  MoveL 9308 to (-40.61, 150.52, 135.08) mm, rotated rx 180 ry 0 rz -180 deg; joints [-126.331, -50.727, -84.518, 62.425, 65.347, -38.616]
  Call Extruder(4.93416)
  MoveL 9309 to (-40.66, 150.21, 135.08) mm, rotated rx 180 ry 0 rz -180 deg; joints [-126.35, -50.704, -84.571, 62.397, 65.348, -38.58]
  MoveL 9310 to (-40.66, 150.21, 135.08) mm, rotated rx 180 ry 0 rz -180 deg; joints [-126.35, -50.704, -84.571, 62.397, 65.348, -38.58]
  Call Extruder(5.09479)
  MoveL 9311 to (-40.71, 149.91, 135.08) mm, rotated rx -180 ry 0 rz 180 deg; joints [-126.369, -50.681, -84.624, 62.368, 65.35, -38.544]
  MoveL 9312 to (-40.71, 149.91, 135.08) mm, rotated rx -180 ry 0 rz 180 deg; joints [-126.369, -50.681, -84.624, 62.368, 65.35, -38.544]
  Call Extruder(5.25470)
  MoveL 9313 to (-40.76, 149.6, 135.08) mm, rotated rx 180 ry 0 rz -180 deg; joints [-126.388, -50.658, -84.676, 62.34, 65.352, -38.509]
  MoveL 9314 to (-40.76, 149.6, 135.08) mm, rotated rx 180 ry 0 rz -180 deg; joints [-126.388, -50.658, -84.676, 62.34, 65.352, -38.509]
  Call Extruder(5.41388)
  MoveL 9315 to (-40.81, 149.3, 135.08) mm, rotated rx 180 ry 0 rz 180 deg; joints [-126.407, -50.634, -84.729, 62.311, 65.354, -38.473]
  MoveL 9316 to (-40.81, 149.3, 135.08) mm, rotated rx 180 ry 0 rz 180 deg; joints [-126.407, -50.634, -84.729, 62.311, 65.354, -38.473]
  Call Extruder(5.57233)
  MoveL 9317 to (-40.86, 148.99, 135.08) mm, rotated rx 180 ry 0 rz -180 deg; joints [-126.426, -50.611, -84.782, 62.283, 65.356, -38.437]
  MoveL 9318 to (-40.86, 148.99, 135.08) mm, rotated rx 180 ry 0 rz -180 deg; joints [-126.426, -50.611, -84.782, 62.283, 65.356, -38.437]
  Call Extruder(5.77120)
  MoveL 9319 to (-40.9, 148.6, 135.08) mm, rotated rx 180 ry 0 rz 180 deg; joints [-126.452, -50.583, -84.847, 62.246, 65.357, -38.393]
  MoveL 9320 to (-40.9, 148.6, 135.08) mm, rotated rx 180 ry 0 rz 180 deg; joints [-126.452, -50.583, -84.847, 62.246, 65.357, -38.393]
  Call Extruder(5.96921)
  MoveL 9321 to (-40.95, 148.22, 135.08) mm, rotated rx 180 ry 0 rz 180 deg; joints [-126.478, -50.554, -84.912, 62.208, 65.358, -38.348]
  MoveL 9322 to (-40.95, 148.22, 135.08) mm, rotated rx 180 ry 0 rz 180 deg; joints [-126.478, -50.554, -84.912, 62.208, 65.358, -38.348]
  Call Extruder(6.16635)
  MoveL 9323 to (-40.99, 147.83, 135.08) mm, rotated rx 180 ry 0 rz -180 deg; joints [-126.504, -50.526, -84.977, 62.171, 65.359, -38.303]
  MoveL 9324 to (-40.99, 147.83, 135.08) mm, rotated rx 180 ry 0 rz -180 deg; joints [-126.504, -50.526, -84.977, 62.171, 65.359, -38.303]
  Call Extruder(6.36262)
  MoveL 9325 to (-41.04, 147.44, 135.08) mm, rotated rx -180 ry 0 rz 180 deg; joints [-126.53, -50.498, -85.041, 62.134, 65.359, -38.258]
  MoveL 9326 to (-41.04, 147.44, 135.08) mm, rotated rx -180 ry 0 rz 180 deg; joints [-126.53, -50.498, -85.041, 62.134, 65.359, -38.258]
  Call Extruder(6.60831)
  MoveL 9327 to (-41.09, 146.95, 135.08) mm, rotated rx 180 ry 0 rz 180 deg; joints [-126.564, -50.462, -85.122, 62.086, 65.359, -38.202]
  MoveL 9328 to (-41.09, 146.95, 135.08) mm, rotated rx 180 ry 0 rz 180 deg; joints [-126.564, -50.462, -85.122, 62.086, 65.359, -38.202]
  Call Extruder(6.90304)
  MoveL 9329 to (-41.13, 146.36, 135.08) mm, rotated rx 180 ry 0 rz 180 deg; joints [-126.607, -50.421, -85.217, 62.028, 65.358, -38.134]
  MoveL 9330 to (-41.13, 146.36, 135.08) mm, rotated rx 180 ry 0 rz 180 deg; joints [-126.607, -50.421, -85.217, 62.028, 65.358, -38.134]
  Call Extruder(7.19644)
  MoveL 9331 to (-41.18, 145.77, 135.08) mm, rotated rx 180 ry 0 rz -180 deg; joints [-126.649, -50.379, -85.313, 61.969, 65.358, -38.067]
  MoveL 9332 to (-41.18, 145.77, 135.08) mm, rotated rx 180 ry 0 rz -180 deg; joints [-126.649, -50.379, -85.313, 61.969, 65.358, -38.067]
  Call Extruder(7.62977)
  MoveL 9333 to (-41.22, 144.9, 135.08) mm, rotated rx -180 ry 0 rz -180 deg; joints [-126.715, -50.318, -85.452, 61.881, 65.354, -37.967]
  MoveL 9334 to (-41.22, 144.9, 135.08) mm, rotated rx -180 ry 0 rz -180 deg; joints [-126.715, -50.318, -85.452, 61.881, 65.354, -37.967]
  Call Extruder(8.20193)
  MoveL 9335 to (-41.27, 143.74, 135.08) mm, rotated rx 180 ry 0 rz 180 deg; joints [-126.804, -50.238, -85.635, 61.762, 65.348, -37.835]
  MoveL 9336 to (-41.27, 143.74, 135.08) mm, rotated rx 180 ry 0 rz 180 deg; joints [-126.804, -50.238, -85.635, 61.762, 65.348, -37.835]
  Call Extruder(8.62976)
  MoveL 9337 to (-41.29, 142.86, 135.08) mm, rotated rx -180 ry 0 rz 180 deg; joints [-126.873, -50.179, -85.77, 61.671, 65.341, -37.736]
  Call Extruder(50.62329)
  MoveL 9338 to (-41.29, 57.14, 135.08) mm, rotated rx 180 ry 0 rz 180 deg; joints [-135.148, -45.231, -97.556, 51.322, 64.612, -28.173]
  MoveL 9339 to (-41.29, 57.14, 135.08) mm, rotated rx 180 ry 0 rz 180 deg; joints [-135.148, -45.231, -97.556, 51.322, 64.612, -28.173]
  Call Extruder(51.33886)
  MoveL 9340 to (-41.25, 55.68, 135.08) mm, rotated rx -180 ry 0 rz 180 deg; joints [-135.318, -45.162, -97.729, 51.117, 64.597, -28.012]
  MoveL 9341 to (-41.25, 55.68, 135.08) mm, rotated rx -180 ry 0 rz 180 deg; joints [-135.318, -45.162, -97.729, 51.117, 64.597, -28.012]
  Call Extruder(51.91360)
  MoveL 9342 to (-41.2, 54.52, 135.08) mm, rotated rx 180 ry 0 rz -180 deg; joints [-135.457, -45.107, -97.865, 50.952, 64.583, -27.884]
  MoveL 9343 to (-41.2, 54.52, 135.08) mm, rotated rx 180 ry 0 rz -180 deg; joints [-135.457, -45.107, -97.865, 50.952, 64.583, -27.884]
  Call Extruder(52.20698)
  MoveL 9344 to (-41.15, 53.93, 135.08) mm, rotated rx 180 ry 0 rz 180 deg; joints [-135.53, -45.081, -97.932, 50.866, 64.574, -27.819]
  MoveL 9345 to (-41.15, 53.93, 135.08) mm, rotated rx 180 ry 0 rz 180 deg; joints [-135.53, -45.081, -97.932, 50.866, 64.574, -27.819]
  Call Extruder(52.50168)
  MoveL 9346 to (-41.11, 53.34, 135.08) mm, rotated rx 180 ry 0 rz -180 deg; joints [-135.603, -45.054, -97.997, 50.779, 64.565, -27.754]
  MoveL 9347 to (-41.11, 53.34, 135.08) mm, rotated rx 180 ry 0 rz -180 deg; joints [-135.603, -45.054, -97.997, 50.779, 64.565, -27.754]
  Call Extruder(52.79772)
  MoveL 9348 to (-41.06, 52.75, 135.08) mm, rotated rx -180 ry 0 rz 180 deg; joints [-135.676, -45.028, -98.063, 50.693, 64.556, -27.689]
  MoveL 9349 to (-41.06, 52.75, 135.08) mm, rotated rx -180 ry 0 rz 180 deg; joints [-135.676, -45.028, -98.063, 50.693, 64.556, -27.689]
  Call Extruder(52.99180)
  MoveL 9350 to (-41.02, 52.37, 135.08) mm, rotated rx -180 ry 0 rz 180 deg; joints [-135.726, -45.012, -98.104, 50.635, 64.549, -27.647]
  MoveL 9351 to (-41.02, 52.37, 135.08) mm, rotated rx -180 ry 0 rz 180 deg; joints [-135.726, -45.012, -98.104, 50.635, 64.549, -27.647]
  Call Extruder(53.18958)
  MoveL 9352 to (-40.97, 51.98, 135.08) mm, rotated rx 180 ry 0 rz -180 deg; joints [-135.776, -44.995, -98.145, 50.577, 64.541, -27.605]
  MoveL 9353 to (-40.97, 51.98, 135.08) mm, rotated rx 180 ry 0 rz -180 deg; joints [-135.776, -44.995, -98.145, 50.577, 64.541, -27.605]
  Call Extruder(53.38824)
  MoveL 9354 to (-40.92, 51.59, 135.08) mm, rotated rx 180 ry 0 rz 180 deg; joints [-135.826, -44.979, -98.187, 50.518, 64.534, -27.562]
  MoveL 9355 to (-40.92, 51.59, 135.08) mm, rotated rx 180 ry 0 rz 180 deg; joints [-135.826, -44.979, -98.187, 50.518, 64.534, -27.562]
  Call Extruder(53.58777)
  MoveL 9356 to (-40.88, 51.2, 135.08) mm, rotated rx 180 ry 0 rz -180 deg; joints [-135.877, -44.963, -98.228, 50.46, 64.526, -27.52]
  MoveL 9357 to (-40.88, 51.2, 135.08) mm, rotated rx 180 ry 0 rz -180 deg; joints [-135.877, -44.963, -98.228, 50.46, 64.526, -27.52]
  Call Extruder(53.76717)
  MoveL 9358 to (-40.83, 50.86, 135.08) mm, rotated rx 180 ry 0 rz -180 deg; joints [-135.922, -44.948, -98.264, 50.407, 64.519, -27.482]
  MoveL 9359 to (-40.83, 50.86, 135.08) mm, rotated rx 180 ry 0 rz -180 deg; joints [-135.922, -44.948, -98.264, 50.407, 64.519, -27.482]
  Call Extruder(53.92635)
  MoveL 9360 to (-40.78, 50.55, 135.08) mm, rotated rx -180 ry 0 rz -180 deg; joints [-135.964, -44.936, -98.295, 50.36, 64.512, -27.449]
  MoveL 9361 to (-40.78, 50.55, 135.08) mm, rotated rx -180 ry 0 rz -180 deg; joints [-135.964, -44.936, -98.295, 50.36, 64.512, -27.449]
  Call Extruder(54.08625)
  MoveL 9362 to (-40.73, 50.24, 135.08) mm, rotated rx -180 ry 0 rz -180 deg; joints [-136.005, -44.924, -98.326, 50.312, 64.504, -27.416]
  MoveL 9363 to (-40.73, 50.24, 135.08) mm, rotated rx -180 ry 0 rz -180 deg; joints [-136.005, -44.924, -98.326, 50.312, 64.504, -27.416]
  Call Extruder(54.24689)
  MoveL 9364 to (-40.69, 49.94, 135.08) mm, rotated rx 180 ry 0 rz -180 deg; joints [-136.046, -44.911, -98.356, 50.265, 64.497, -27.382]
  MoveL 9365 to (-40.69, 49.94, 135.08) mm, rotated rx 180 ry 0 rz -180 deg; joints [-136.046, -44.911, -98.356, 50.265, 64.497, -27.382]
  Call Extruder(54.40825)
  MoveL 9366 to (-40.64, 49.63, 135.08) mm, rotated rx 180 ry 0 rz 180 deg; joints [-136.087, -44.899, -98.387, 50.218, 64.49, -27.349]
  MoveL 9367 to (-40.64, 49.63, 135.08) mm, rotated rx 180 ry 0 rz 180 deg; joints [-136.087, -44.899, -98.387, 50.218, 64.49, -27.349]
  Call Extruder(54.57034)
  MoveL 9368 to (-40.59, 49.33, 135.08) mm, rotated rx 180 ry 0 rz -180 deg; joints [-136.128, -44.887, -98.418, 50.17, 64.483, -27.316]
  MoveL 9369 to (-40.59, 49.33, 135.08) mm, rotated rx 180 ry 0 rz -180 deg; joints [-136.128, -44.887, -98.418, 50.17, 64.483, -27.316]
  Call Extruder(54.71853)
  MoveL 9370 to (-40.54, 49.05, 135.08) mm, rotated rx -180 ry 0 rz 180 deg; joints [-136.166, -44.876, -98.445, 50.127, 64.476, -27.286]
  MoveL 9371 to (-40.54, 49.05, 135.08) mm, rotated rx -180 ry 0 rz 180 deg; joints [-136.166, -44.876, -98.445, 50.127, 64.476, -27.286]
  Call Extruder(54.85276)
  MoveL 9372 to (-40.49, 48.8, 135.08) mm, rotated rx 180 ry 0 rz -180 deg; joints [-136.201, -44.867, -98.468, 50.087, 64.469, -27.259]
  MoveL 9373 to (-40.49, 48.8, 135.08) mm, rotated rx 180 ry 0 rz -180 deg; joints [-136.201, -44.867, -98.468, 50.087, 64.469, -27.259]
  Call Extruder(54.98760)
  MoveL 9374 to (-40.44, 48.55, 135.08) mm, rotated rx 180 ry 0 rz -180 deg; joints [-136.236, -44.858, -98.492, 50.048, 64.462, -27.232]
  MoveL 9375 to (-40.44, 48.55, 135.08) mm, rotated rx 180 ry 0 rz -180 deg; joints [-136.236, -44.858, -98.492, 50.048, 64.462, -27.232]
  Call Extruder(55.12305)
  MoveL 9376 to (-40.39, 48.3, 135.08) mm, rotated rx 180 ry 0 rz 180 deg; joints [-136.271, -44.848, -98.516, 50.008, 64.456, -27.205]
  MoveL 9377 to (-40.39, 48.3, 135.08) mm, rotated rx 180 ry 0 rz 180 deg; joints [-136.271, -44.848, -98.516, 50.008, 64.456, -27.205]
  Call Extruder(55.25911)
  MoveL 9378 to (-40.34, 48.05, 135.08) mm, rotated rx -180 ry 0 rz 180 deg; joints [-136.306, -44.839, -98.539, 49.969, 64.449, -27.178]
  MoveL 9379 to (-40.34, 48.05, 135.08) mm, rotated rx -180 ry 0 rz 180 deg; joints [-136.306, -44.839, -98.539, 49.969, 64.449, -27.178]
  Call Extruder(55.39578)
  MoveL 9380 to (-40.29, 47.8, 135.08) mm, rotated rx -180 ry 0 rz -180 deg; joints [-136.341, -44.829, -98.563, 49.929, 64.442, -27.151]
  MoveL 9381 to (-40.29, 47.8, 135.08) mm, rotated rx -180 ry 0 rz -180 deg; joints [-136.341, -44.829, -98.563, 49.929, 64.442, -27.151]
  Call Extruder(55.53306)
  MoveL 9382 to (-40.24, 47.55, 135.08) mm, rotated rx -180 ry 0 rz -180 deg; joints [-136.376, -44.82, -98.586, 49.889, 64.435, -27.124]
  MoveL 9383 to (-40.24, 47.55, 135.08) mm, rotated rx -180 ry 0 rz -180 deg; joints [-136.376, -44.82, -98.586, 49.889, 64.435, -27.124]
  Call Extruder(55.65874)
  MoveL 9384 to (-40.2, 47.33, 135.08) mm, rotated rx 180 ry 0 rz 180 deg; joints [-136.408, -44.812, -98.607, 49.853, 64.429, -27.1]
  MoveL 9385 to (-40.2, 47.33, 135.08) mm, rotated rx 180 ry 0 rz 180 deg; joints [-136.408, -44.812, -98.607, 49.853, 64.429, -27.1]
  Call Extruder(55.77269)
  MoveL 9386 to (-40.15, 47.12, 135.08) mm, rotated rx 180 ry 0 rz -180 deg; joints [-136.437, -44.804, -98.626, 49.82, 64.423, -27.078]
  MoveL 9387 to (-40.15, 47.12, 135.08) mm, rotated rx 180 ry 0 rz -180 deg; joints [-136.437, -44.804, -98.626, 49.82, 64.423, -27.078]
  Call Extruder(55.88710)
  MoveL 9388 to (-40.11, 46.92, 135.08) mm, rotated rx 180 ry 0 rz 180 deg; joints [-136.466, -44.797, -98.645, 49.787, 64.417, -27.056]
  MoveL 9389 to (-40.11, 46.92, 135.08) mm, rotated rx 180 ry 0 rz 180 deg; joints [-136.466, -44.797, -98.645, 49.787, 64.417, -27.056]
  Call Extruder(56.00196)
  MoveL 9390 to (-40.06, 46.72, 135.08) mm, rotated rx 180 ry 0 rz 180 deg; joints [-136.495, -44.789, -98.664, 49.754, 64.411, -27.034]
  MoveL 9391 to (-40.06, 46.72, 135.08) mm, rotated rx 180 ry 0 rz 180 deg; joints [-136.495, -44.789, -98.664, 49.754, 64.411, -27.034]
  Call Extruder(56.11727)
  MoveL 9392 to (-40.02, 46.51, 135.08) mm, rotated rx -180 ry 0 rz -180 deg; joints [-136.525, -44.782, -98.682, 49.721, 64.405, -27.012]
  MoveL 9393 to (-40.02, 46.51, 135.08) mm, rotated rx -180 ry 0 rz -180 deg; joints [-136.525, -44.782, -98.682, 49.721, 64.405, -27.012]
  Call Extruder(56.24665)
  MoveL 9394 to (-39.95, 46.29, 135.08) mm, rotated rx 180 ry 0 rz -180 deg; joints [-136.559, -44.775, -98.701, 49.684, 64.397, -26.988]
  MoveL 9395 to (-39.95, 46.29, 135.08) mm, rotated rx 180 ry 0 rz -180 deg; joints [-136.559, -44.775, -98.701, 49.684, 64.397, -26.988]
  Call Extruder(56.37660)
  MoveL 9396 to (-39.88, 46.06, 135.08) mm, rotated rx 180 ry 0 rz -180 deg; joints [-136.593, -44.768, -98.719, 49.646, 64.388, -26.964]
  MoveL 9397 to (-39.88, 46.06, 135.08) mm, rotated rx 180 ry 0 rz -180 deg; joints [-136.593, -44.768, -98.719, 49.646, 64.388, -26.964]
  Call Extruder(56.50711)
  MoveL 9398 to (-39.81, 45.84, 135.08) mm, rotated rx 180 ry 0 rz 180 deg; joints [-136.627, -44.76, -98.737, 49.608, 64.38, -26.941]
  MoveL 9399 to (-39.81, 45.84, 135.08) mm, rotated rx 180 ry 0 rz 180 deg; joints [-136.627, -44.76, -98.737, 49.608, 64.38, -26.941]
  Call Extruder(56.63818)
  MoveL 9400 to (-39.75, 45.62, 135.08) mm, rotated rx -180 ry 0 rz 180 deg; joints [-136.661, -44.753, -98.755, 49.57, 64.371, -26.917]
  MoveL 9401 to (-39.75, 45.62, 135.08) mm, rotated rx -180 ry 0 rz 180 deg; joints [-136.661, -44.753, -98.755, 49.57, 64.371, -26.917]
  Call Extruder(56.75983)
  MoveL 9402 to (-39.68, 45.41, 135.08) mm, rotated rx 180 ry 0 rz -180 deg; joints [-136.693, -44.747, -98.771, 49.535, 64.363, -26.895]
  MoveL 9403 to (-39.68, 45.41, 135.08) mm, rotated rx 180 ry 0 rz -180 deg; joints [-136.693, -44.747, -98.771, 49.535, 64.363, -26.895]
  Call Extruder(56.87195)
  MoveL 9404 to (-39.62, 45.22, 135.08) mm, rotated rx 180 ry 0 rz 180 deg; joints [-136.722, -44.741, -98.786, 49.503, 64.356, -26.875]
  MoveL 9405 to (-39.62, 45.22, 135.08) mm, rotated rx 180 ry 0 rz 180 deg; joints [-136.722, -44.741, -98.786, 49.503, 64.356, -26.875]
  Call Extruder(56.98452)
  MoveL 9406 to (-39.56, 45.03, 135.08) mm, rotated rx 180 ry 0 rz -180 deg; joints [-136.751, -44.735, -98.8, 49.471, 64.348, -26.855]
  MoveL 9407 to (-39.56, 45.03, 135.08) mm, rotated rx 180 ry 0 rz -180 deg; joints [-136.751, -44.735, -98.8, 49.471, 64.348, -26.855]
  Call Extruder(57.09753)
  MoveL 9408 to (-39.5, 44.85, 135.08) mm, rotated rx 180 ry 0 rz -180 deg; joints [-136.781, -44.73, -98.815, 49.439, 64.341, -26.835]
  MoveL 9409 to (-39.5, 44.85, 135.08) mm, rotated rx 180 ry 0 rz -180 deg; joints [-136.781, -44.73, -98.815, 49.439, 64.341, -26.835]
  Call Extruder(57.21099)
  MoveL 9410 to (-39.44, 44.66, 135.08) mm, rotated rx 180 ry 0 rz -180 deg; joints [-136.81, -44.724, -98.829, 49.406, 64.333, -26.815]
  MoveL 9411 to (-39.44, 44.66, 135.08) mm, rotated rx 180 ry 0 rz -180 deg; joints [-136.81, -44.724, -98.829, 49.406, 64.333, -26.815]
  Call Extruder(57.35863)
  MoveL 9412 to (-39.35, 44.42, 135.08) mm, rotated rx 180 ry 0 rz -180 deg; joints [-136.849, -44.717, -98.846, 49.364, 64.322, -26.79]
  MoveL 9413 to (-39.35, 44.42, 135.08) mm, rotated rx 180 ry 0 rz -180 deg; joints [-136.849, -44.717, -98.846, 49.364, 64.322, -26.79]
  Call Extruder(57.54097)
  MoveL 9414 to (-39.23, 44.12, 135.08) mm, rotated rx 180 ry 0 rz 180 deg; joints [-136.898, -44.709, -98.865, 49.312, 64.308, -26.759]
  MoveL 9415 to (-39.23, 44.12, 135.08) mm, rotated rx 180 ry 0 rz 180 deg; joints [-136.898, -44.709, -98.865, 49.312, 64.308, -26.759]
  Call Extruder(57.72406)
  MoveL 9416 to (-39.11, 43.83, 135.08) mm, rotated rx 180 ry 0 rz -180 deg; joints [-136.946, -44.702, -98.885, 49.26, 64.294, -26.728]
  MoveL 9417 to (-39.11, 43.83, 135.08) mm, rotated rx 180 ry 0 rz -180 deg; joints [-136.946, -44.702, -98.885, 49.26, 64.294, -26.728]
  Call Extruder(57.88175)
  MoveL 9418 to (-39, 43.58, 135.08) mm, rotated rx 180 ry 0 rz -180 deg; joints [-136.988, -44.696, -98.901, 49.215, 64.281, -26.702]
  MoveL 9419 to (-39, 43.58, 135.08) mm, rotated rx 180 ry 0 rz -180 deg; joints [-136.988, -44.696, -98.901, 49.215, 64.281, -26.702]
  Call Extruder(58.04004)
  MoveL 9420 to (-38.89, 43.33, 135.08) mm, rotated rx -180 ry 0 rz 180 deg; joints [-137.029, -44.689, -98.916, 49.17, 64.269, -26.676]
  MoveL 9421 to (-38.89, 43.33, 135.08) mm, rotated rx -180 ry 0 rz 180 deg; joints [-137.029, -44.689, -98.916, 49.17, 64.269, -26.676]
  Call Extruder(58.22206)
  MoveL 9422 to (-38.75, 43.06, 135.08) mm, rotated rx 180 ry 0 rz -180 deg; joints [-137.078, -44.684, -98.931, 49.118, 64.253, -26.648]
  MoveL 9423 to (-38.75, 43.06, 135.08) mm, rotated rx 180 ry 0 rz -180 deg; joints [-137.078, -44.684, -98.931, 49.118, 64.253, -26.648]
  Call Extruder(58.42862)
  MoveL 9424 to (-38.57, 42.75, 135.08) mm, rotated rx 180 ry 0 rz -180 deg; joints [-137.135, -44.678, -98.945, 49.059, 64.233, -26.617]
  MoveL 9425 to (-38.57, 42.75, 135.08) mm, rotated rx 180 ry 0 rz -180 deg; joints [-137.135, -44.678, -98.945, 49.059, 64.233, -26.617]
  Call Extruder(58.63595)
  MoveL 9426 to (-38.4, 42.45, 135.08) mm, rotated rx -180 ry 0 rz -180 deg; joints [-137.191, -44.673, -98.958, 49.001, 64.213, -26.586]
  MoveL 9427 to (-38.4, 42.45, 135.08) mm, rotated rx -180 ry 0 rz -180 deg; joints [-137.191, -44.673, -98.958, 49.001, 64.213, -26.586]
  Call Extruder(58.84406)
  MoveL 9428 to (-38.22, 42.15, 135.08) mm, rotated rx 180 ry 0 rz 180 deg; joints [-137.247, -44.668, -98.971, 48.942, 64.193, -26.555]
  MoveL 9429 to (-38.22, 42.15, 135.08) mm, rotated rx 180 ry 0 rz 180 deg; joints [-137.247, -44.668, -98.971, 48.942, 64.193, -26.555]
  Call Extruder(58.96178)
  MoveL 9430 to (-38.12, 41.98, 135.08) mm, rotated rx 180 ry 0 rz 180 deg; joints [-137.279, -44.665, -98.979, 48.909, 64.182, -26.537]
  MoveL 9431 to (-38.12, 41.98, 135.08) mm, rotated rx 180 ry 0 rz 180 deg; joints [-137.279, -44.665, -98.979, 48.909, 64.182, -26.537]
  Call Extruder(59.29462)
  MoveL 9432 to (-37.8, 41.52, 135.08) mm, rotated rx -180 ry 0 rz 180 deg; joints [-137.37, -44.66, -98.99, 48.816, 64.146, -26.492]
  MoveL 9433 to (-37.8, 41.52, 135.08) mm, rotated rx -180 ry 0 rz 180 deg; joints [-137.37, -44.66, -98.99, 48.816, 64.146, -26.492]
  Call Extruder(59.62865)
  MoveL 9434 to (-37.47, 41.07, 135.08) mm, rotated rx 180 ry 0 rz 180 deg; joints [-137.461, -44.656, -99.001, 48.723, 64.11, -26.447]
  MoveL 9435 to (-37.47, 41.07, 135.08) mm, rotated rx 180 ry 0 rz 180 deg; joints [-137.461, -44.656, -99.001, 48.723, 64.11, -26.447]
  Call Extruder(59.79624)
  MoveL 9436 to (-37.3, 40.85, 135.08) mm, rotated rx 180 ry 0 rz 180 deg; joints [-137.506, -44.654, -99.007, 48.676, 64.092, -26.424]
  Call Extruder(60.62555)
  MoveL 9437 to (-36.39, 39.81, 135.08) mm, rotated rx 180 ry 0 rz -180 deg; joints [-137.733, -44.652, -99.011, 48.449, 63.993, -26.323]
  Call Extruder(61.25663)
  MoveL 9438 to (-35.6, 39.11, 135.08) mm, rotated rx 180 ry 0 rz 180 deg; joints [-137.904, -44.66, -98.991, 48.283, 63.909, -26.258]
  MoveL 9439 to (-35.6, 39.11, 135.08) mm, rotated rx 180 ry 0 rz 180 deg; joints [-137.904, -44.66, -98.991, 48.283, 63.909, -26.258]
  Call Extruder(61.45419)
  MoveL 9440 to (-35.35, 38.9, 135.08) mm, rotated rx 180 ry 0 rz -180 deg; joints [-137.958, -44.663, -98.984, 48.231, 63.882, -26.238]
  Call Extruder(61.78821)
  MoveL 9441 to (-34.9, 38.57, 135.08) mm, rotated rx 180 ry 0 rz 180 deg; joints [-138.048, -44.671, -98.964, 48.145, 63.834, -26.209]
  MoveL 9442 to (-34.9, 38.57, 135.08) mm, rotated rx 180 ry 0 rz 180 deg; joints [-138.048, -44.671, -98.964, 48.145, 63.834, -26.209]
  Call Extruder(62.12104)
  MoveL 9443 to (-34.45, 38.24, 135.08) mm, rotated rx 180 ry 0 rz 180 deg; joints [-138.137, -44.679, -98.944, 48.06, 63.787, -26.179]
  MoveL 9444 to (-34.45, 38.24, 135.08) mm, rotated rx 180 ry 0 rz 180 deg; joints [-138.137, -44.679, -98.944, 48.06, 63.787, -26.179]
  Call Extruder(62.30029)
  MoveL 9445 to (-34.21, 38.07, 135.08) mm, rotated rx 180 ry 0 rz 180 deg; joints [-138.185, -44.683, -98.932, 48.015, 63.761, -26.164]
  MoveL 9446 to (-34.21, 38.07, 135.08) mm, rotated rx 180 ry 0 rz 180 deg; joints [-138.185, -44.683, -98.932, 48.015, 63.761, -26.164]
  Call Extruder(62.50840)
  MoveL 9447 to (-33.9, 37.89, 135.08) mm, rotated rx 180 ry 0 rz -180 deg; joints [-138.24, -44.69, -98.914, 47.964, 63.729, -26.149]
  MoveL 9448 to (-33.9, 37.89, 135.08) mm, rotated rx 180 ry 0 rz -180 deg; joints [-138.24, -44.69, -98.914, 47.964, 63.729, -26.149]
  Call Extruder(62.71573)
  MoveL 9449 to (-33.6, 37.71, 135.08) mm, rotated rx -180 ry 0 rz 180 deg; joints [-138.295, -44.698, -98.895, 47.914, 63.697, -26.134]
  MoveL 9450 to (-33.6, 37.71, 135.08) mm, rotated rx -180 ry 0 rz 180 deg; joints [-138.295, -44.698, -98.895, 47.914, 63.697, -26.134]
  Call Extruder(62.92229)
  MoveL 9451 to (-33.29, 37.54, 135.08) mm, rotated rx 180 ry 0 rz 180 deg; joints [-138.349, -44.706, -98.876, 47.863, 63.666, -26.119]
  MoveL 9452 to (-33.29, 37.54, 135.08) mm, rotated rx 180 ry 0 rz 180 deg; joints [-138.349, -44.706, -98.876, 47.863, 63.666, -26.119]
  Call Extruder(63.12806)
  MoveL 9453 to (-32.99, 37.36, 135.08) mm, rotated rx 180 ry 0 rz 180 deg; joints [-138.404, -44.713, -98.856, 47.813, 63.634, -26.105]
  MoveL 9454 to (-32.99, 37.36, 135.08) mm, rotated rx 180 ry 0 rz 180 deg; joints [-138.404, -44.713, -98.856, 47.813, 63.634, -26.105]
  Call Extruder(63.28636)
  MoveL 9455 to (-32.74, 37.26, 135.08) mm, rotated rx -180 ry 0 rz -180 deg; joints [-138.444, -44.721, -98.836, 47.777, 63.608, -26.097]
  MoveL 9456 to (-32.74, 37.26, 135.08) mm, rotated rx -180 ry 0 rz -180 deg; joints [-138.444, -44.721, -98.836, 47.777, 63.608, -26.097]
  Call Extruder(63.44406)
  MoveL 9457 to (-32.49, 37.15, 135.08) mm, rotated rx 180 ry 0 rz 180 deg; joints [-138.484, -44.729, -98.816, 47.741, 63.582, -26.089]
  MoveL 9458 to (-32.49, 37.15, 135.08) mm, rotated rx 180 ry 0 rz 180 deg; joints [-138.484, -44.729, -98.816, 47.741, 63.582, -26.089]
  Call Extruder(63.61415)
  MoveL 9459 to (-32.22, 37.03, 135.08) mm, rotated rx 180 ry 0 rz 180 deg; joints [-138.527, -44.738, -98.795, 47.703, 63.554, -26.081]
  MoveL 9460 to (-32.22, 37.03, 135.08) mm, rotated rx 180 ry 0 rz 180 deg; joints [-138.527, -44.738, -98.795, 47.703, 63.554, -26.081]
  Call Extruder(63.79648)
  MoveL 9461 to (-31.93, 36.91, 135.08) mm, rotated rx -180 ry 0 rz -180 deg; joints [-138.574, -44.747, -98.771, 47.661, 63.524, -26.072]
  MoveL 9462 to (-31.93, 36.91, 135.08) mm, rotated rx -180 ry 0 rz -180 deg; joints [-138.574, -44.747, -98.771, 47.661, 63.524, -26.072]
  Call Extruder(63.97805)
  MoveL 9463 to (-31.64, 36.79, 135.08) mm, rotated rx -180 ry 0 rz 180 deg; joints [-138.62, -44.757, -98.747, 47.62, 63.494, -26.063]
  MoveL 9464 to (-31.64, 36.79, 135.08) mm, rotated rx -180 ry 0 rz 180 deg; joints [-138.62, -44.757, -98.747, 47.62, 63.494, -26.063]
  Call Extruder(64.09151)
  MoveL 9465 to (-31.45, 36.73, 135.08) mm, rotated rx 180 ry 0 rz -180 deg; joints [-138.648, -44.763, -98.729, 47.596, 63.475, -26.059]
  MoveL 9466 to (-31.45, 36.73, 135.08) mm, rotated rx 180 ry 0 rz -180 deg; joints [-138.648, -44.763, -98.729, 47.596, 63.475, -26.059]
  Call Extruder(64.20453)
  MoveL 9467 to (-31.26, 36.67, 135.08) mm, rotated rx -180 ry 0 rz -180 deg; joints [-138.676, -44.77, -98.712, 47.572, 63.455, -26.055]
  MoveL 9468 to (-31.26, 36.67, 135.08) mm, rotated rx -180 ry 0 rz -180 deg; joints [-138.676, -44.77, -98.712, 47.572, 63.455, -26.055]
  Call Extruder(64.31709)
  MoveL 9469 to (-31.07, 36.61, 135.08) mm, rotated rx 180 ry 0 rz 180 deg; joints [-138.704, -44.777, -98.694, 47.548, 63.436, -26.052]
  MoveL 9470 to (-31.07, 36.61, 135.08) mm, rotated rx 180 ry 0 rz 180 deg; joints [-138.704, -44.777, -98.694, 47.548, 63.436, -26.052]
  Call Extruder(64.42922)
  MoveL 9471 to (-30.88, 36.55, 135.08) mm, rotated rx 180 ry 0 rz -180 deg; joints [-138.732, -44.784, -98.677, 47.524, 63.417, -26.048]
  MoveL 9472 to (-30.88, 36.55, 135.08) mm, rotated rx 180 ry 0 rz -180 deg; joints [-138.732, -44.784, -98.677, 47.524, 63.417, -26.048]
  Call Extruder(64.54090)
  MoveL 9473 to (-30.69, 36.49, 135.08) mm, rotated rx 180 ry 0 rz -180 deg; joints [-138.759, -44.791, -98.659, 47.5, 63.397, -26.044]
  MoveL 9474 to (-30.69, 36.49, 135.08) mm, rotated rx 180 ry 0 rz -180 deg; joints [-138.759, -44.791, -98.659, 47.5, 63.397, -26.044]
  Call Extruder(64.67197)
  MoveL 9475 to (-30.47, 36.42, 135.08) mm, rotated rx -180 ry 0 rz -180 deg; joints [-138.792, -44.8, -98.638, 47.472, 63.374, -26.04]
  MoveL 9476 to (-30.47, 36.42, 135.08) mm, rotated rx -180 ry 0 rz -180 deg; joints [-138.792, -44.8, -98.638, 47.472, 63.374, -26.04]
  Call Extruder(64.80248)
  MoveL 9477 to (-30.25, 36.35, 135.08) mm, rotated rx 180 ry 0 rz -180 deg; joints [-138.824, -44.808, -98.616, 47.444, 63.351, -26.036]
  MoveL 9478 to (-30.25, 36.35, 135.08) mm, rotated rx 180 ry 0 rz -180 deg; joints [-138.824, -44.808, -98.616, 47.444, 63.351, -26.036]
  Call Extruder(64.93242)
  MoveL 9479 to (-30.02, 36.28, 135.08) mm, rotated rx 180 ry 0 rz -180 deg; joints [-138.856, -44.817, -98.595, 47.417, 63.329, -26.032]
  MoveL 9480 to (-30.02, 36.28, 135.08) mm, rotated rx 180 ry 0 rz -180 deg; joints [-138.856, -44.817, -98.595, 47.417, 63.329, -26.032]
  Call Extruder(65.06180)
  MoveL 9481 to (-29.8, 36.22, 135.08) mm, rotated rx 180 ry 0 rz -180 deg; joints [-138.889, -44.825, -98.574, 47.389, 63.306, -26.028]
  MoveL 9482 to (-29.8, 36.22, 135.08) mm, rotated rx 180 ry 0 rz -180 deg; joints [-138.889, -44.825, -98.574, 47.389, 63.306, -26.028]
  Call Extruder(65.18377)
  MoveL 9483 to (-29.59, 36.16, 135.08) mm, rotated rx 180 ry 0 rz 180 deg; joints [-138.919, -44.834, -98.552, 47.364, 63.284, -26.025]
  MoveL 9484 to (-29.59, 36.16, 135.08) mm, rotated rx 180 ry 0 rz 180 deg; joints [-138.919, -44.834, -98.552, 47.364, 63.284, -26.025]
  Call Extruder(65.29861)
  MoveL 9485 to (-29.38, 36.12, 135.08) mm, rotated rx 180 ry 0 rz 180 deg; joints [-138.946, -44.842, -98.53, 47.341, 63.263, -26.024]
  MoveL 9486 to (-29.38, 36.12, 135.08) mm, rotated rx 180 ry 0 rz 180 deg; joints [-138.946, -44.842, -98.53, 47.341, 63.263, -26.024]
  Call Extruder(65.41301)
  MoveL 9487 to (-29.18, 36.07, 135.08) mm, rotated rx -180 ry 0 rz 180 deg; joints [-138.973, -44.851, -98.509, 47.318, 63.242, -26.022]
  MoveL 9488 to (-29.18, 36.07, 135.08) mm, rotated rx -180 ry 0 rz 180 deg; joints [-138.973, -44.851, -98.509, 47.318, 63.242, -26.022]
  Call Extruder(65.52695)
  MoveL 9489 to (-28.97, 36.03, 135.08) mm, rotated rx -180 ry 0 rz -180 deg; joints [-139, -44.859, -98.487, 47.296, 63.221, -26.021]
  MoveL 9490 to (-28.97, 36.03, 135.08) mm, rotated rx -180 ry 0 rz -180 deg; joints [-139, -44.859, -98.487, 47.296, 63.221, -26.021]
  Call Extruder(65.64044)
  MoveL 9491 to (-28.77, 35.98, 135.08) mm, rotated rx 180 ry 0 rz 180 deg; joints [-139.028, -44.868, -98.466, 47.273, 63.201, -26.019]
  MoveL 9492 to (-28.77, 35.98, 135.08) mm, rotated rx 180 ry 0 rz 180 deg; joints [-139.028, -44.868, -98.466, 47.273, 63.201, -26.019]
  Call Extruder(65.77772)
  MoveL 9493 to (-28.52, 35.93, 135.08) mm, rotated rx 180 ry 0 rz 180 deg; joints [-139.06, -44.879, -98.439, 47.246, 63.175, -26.017]
  MoveL 9494 to (-28.52, 35.93, 135.08) mm, rotated rx 180 ry 0 rz 180 deg; joints [-139.06, -44.879, -98.439, 47.246, 63.175, -26.017]
  Call Extruder(65.91440)
  MoveL 9495 to (-28.27, 35.88, 135.08) mm, rotated rx 180 ry 0 rz 180 deg; joints [-139.093, -44.889, -98.412, 47.219, 63.15, -26.016]
  MoveL 9496 to (-28.27, 35.88, 135.08) mm, rotated rx 180 ry 0 rz 180 deg; joints [-139.093, -44.889, -98.412, 47.219, 63.15, -26.016]
  Call Extruder(66.05046)
  MoveL 9497 to (-28.02, 35.83, 135.08) mm, rotated rx -180 ry 0 rz -180 deg; joints [-139.126, -44.9, -98.385, 47.193, 63.125, -26.015]
  MoveL 9498 to (-28.02, 35.83, 135.08) mm, rotated rx -180 ry 0 rz -180 deg; joints [-139.126, -44.9, -98.385, 47.193, 63.125, -26.015]
  Call Extruder(66.18591)
  MoveL 9499 to (-27.77, 35.78, 135.08) mm, rotated rx 180 ry 0 rz -180 deg; joints [-139.158, -44.911, -98.358, 47.166, 63.099, -26.013]
  MoveL 9500 to (-27.77, 35.78, 135.08) mm, rotated rx 180 ry 0 rz -180 deg; joints [-139.158, -44.911, -98.358, 47.166, 63.099, -26.013]
  Call Extruder(66.32075)
  MoveL 9501 to (-27.52, 35.73, 135.08) mm, rotated rx 180 ry 0 rz 180 deg; joints [-139.191, -44.922, -98.331, 47.139, 63.074, -26.012]
  MoveL 9502 to (-27.52, 35.73, 135.08) mm, rotated rx 180 ry 0 rz 180 deg; joints [-139.191, -44.922, -98.331, 47.139, 63.074, -26.012]
  Call Extruder(66.45498)
  MoveL 9503 to (-27.27, 35.68, 135.08) mm, rotated rx -180 ry 0 rz 180 deg; joints [-139.223, -44.932, -98.304, 47.112, 63.049, -26.01]
  MoveL 9504 to (-27.27, 35.68, 135.08) mm, rotated rx -180 ry 0 rz 180 deg; joints [-139.223, -44.932, -98.304, 47.112, 63.049, -26.01]
  Call Extruder(66.58860)
  MoveL 9505 to (-27.03, 35.63, 135.08) mm, rotated rx -180 ry 0 rz 180 deg; joints [-139.256, -44.943, -98.276, 47.086, 63.023, -26.009]
  MoveL 9506 to (-27.03, 35.63, 135.08) mm, rotated rx -180 ry 0 rz 180 deg; joints [-139.256, -44.943, -98.276, 47.086, 63.023, -26.009]
  Call Extruder(66.75070)
  MoveL 9507 to (-26.72, 35.59, 135.08) mm, rotated rx 180 ry 0 rz 180 deg; joints [-139.294, -44.957, -98.242, 47.055, 62.992, -26.008]
  MoveL 9508 to (-26.72, 35.59, 135.08) mm, rotated rx 180 ry 0 rz 180 deg; joints [-139.294, -44.957, -98.242, 47.055, 62.992, -26.008]
  Call Extruder(66.91207)
  MoveL 9509 to (-26.41, 35.54, 135.08) mm, rotated rx 180 ry 0 rz 180 deg; joints [-139.332, -44.971, -98.207, 47.024, 62.961, -26.008]
  MoveL 9510 to (-26.41, 35.54, 135.08) mm, rotated rx 180 ry 0 rz 180 deg; joints [-139.332, -44.971, -98.207, 47.024, 62.961, -26.008]
  Call Extruder(67.07271)
  MoveL 9511 to (-26.11, 35.49, 135.08) mm, rotated rx 180 ry 0 rz -180 deg; joints [-139.371, -44.985, -98.172, 46.993, 62.93, -26.008]
  MoveL 9512 to (-26.11, 35.49, 135.08) mm, rotated rx 180 ry 0 rz -180 deg; joints [-139.371, -44.985, -98.172, 46.993, 62.93, -26.008]
  Call Extruder(67.23263)
  MoveL 9513 to (-25.8, 35.44, 135.08) mm, rotated rx 180 ry 0 rz -180 deg; joints [-139.409, -44.998, -98.138, 46.963, 62.899, -26.007]
  MoveL 9514 to (-25.8, 35.44, 135.08) mm, rotated rx 180 ry 0 rz -180 deg; joints [-139.409, -44.998, -98.138, 46.963, 62.899, -26.007]
  Call Extruder(67.39181)
  MoveL 9515 to (-25.5, 35.39, 135.08) mm, rotated rx -180 ry 0 rz 180 deg; joints [-139.447, -45.012, -98.103, 46.932, 62.868, -26.007]
  MoveL 9516 to (-25.5, 35.39, 135.08) mm, rotated rx -180 ry 0 rz 180 deg; joints [-139.447, -45.012, -98.103, 46.932, 62.868, -26.007]
  Call Extruder(67.55027)
  MoveL 9517 to (-25.19, 35.34, 135.08) mm, rotated rx 180 ry 0 rz 180 deg; joints [-139.485, -45.026, -98.068, 46.901, 62.837, -26.007]
  MoveL 9518 to (-25.19, 35.34, 135.08) mm, rotated rx 180 ry 0 rz 180 deg; joints [-139.485, -45.026, -98.068, 46.901, 62.837, -26.007]
  Call Extruder(67.74915)
  MoveL 9519 to (-24.8, 35.3, 135.08) mm, rotated rx 180 ry 0 rz -180 deg; joints [-139.531, -45.045, -98.022, 46.865, 62.798, -26.008]
  MoveL 9520 to (-24.8, 35.3, 135.08) mm, rotated rx 180 ry 0 rz -180 deg; joints [-139.531, -45.045, -98.022, 46.865, 62.798, -26.008]
  Call Extruder(67.94716)
  MoveL 9521 to (-24.42, 35.25, 135.08) mm, rotated rx 180 ry 0 rz 180 deg; joints [-139.577, -45.063, -97.976, 46.829, 62.759, -26.009]
  MoveL 9522 to (-24.42, 35.25, 135.08) mm, rotated rx 180 ry 0 rz 180 deg; joints [-139.577, -45.063, -97.976, 46.829, 62.759, -26.009]
  Call Extruder(68.14430)
  MoveL 9523 to (-24.03, 35.21, 135.08) mm, rotated rx 180 ry 0 rz 180 deg; joints [-139.624, -45.081, -97.93, 46.792, 62.72, -26.011]
  MoveL 9524 to (-24.03, 35.21, 135.08) mm, rotated rx 180 ry 0 rz 180 deg; joints [-139.624, -45.081, -97.93, 46.792, 62.72, -26.011]
  Call Extruder(68.34057)
  MoveL 9525 to (-23.64, 35.16, 135.08) mm, rotated rx -180 ry 0 rz 180 deg; joints [-139.67, -45.1, -97.884, 46.756, 62.68, -26.012]
  MoveL 9526 to (-23.64, 35.16, 135.08) mm, rotated rx -180 ry 0 rz 180 deg; joints [-139.67, -45.1, -97.884, 46.756, 62.68, -26.012]
  Call Extruder(68.58626)
  MoveL 9527 to (-23.15, 35.11, 135.08) mm, rotated rx 180 ry 0 rz -180 deg; joints [-139.726, -45.124, -97.824, 46.712, 62.631, -26.015]
  MoveL 9528 to (-23.15, 35.11, 135.08) mm, rotated rx 180 ry 0 rz -180 deg; joints [-139.726, -45.124, -97.824, 46.712, 62.631, -26.015]
  Call Extruder(68.88099)
  MoveL 9529 to (-22.56, 35.07, 135.08) mm, rotated rx 180 ry 0 rz -180 deg; joints [-139.793, -45.153, -97.751, 46.661, 62.572, -26.02]
  MoveL 9530 to (-22.56, 35.07, 135.08) mm, rotated rx 180 ry 0 rz -180 deg; joints [-139.793, -45.153, -97.751, 46.661, 62.572, -26.02]
  Call Extruder(69.17439)
  MoveL 9531 to (-21.97, 35.02, 135.08) mm, rotated rx 180 ry 0 rz 180 deg; joints [-139.86, -45.182, -97.678, 46.61, 62.512, -26.024]
  MoveL 9532 to (-21.97, 35.02, 135.08) mm, rotated rx 180 ry 0 rz 180 deg; joints [-139.86, -45.182, -97.678, 46.61, 62.512, -26.024]
  Call Extruder(69.60772)
  MoveL 9533 to (-21.1, 34.98, 135.08) mm, rotated rx 180 ry 0 rz 180 deg; joints [-139.956, -45.227, -97.566, 46.538, 62.424, -26.034]
  MoveL 9534 to (-21.1, 34.98, 135.08) mm, rotated rx 180 ry 0 rz 180 deg; joints [-139.956, -45.227, -97.566, 46.538, 62.424, -26.034]
  Call Extruder(70.17988)
  MoveL 9535 to (-19.94, 34.93, 135.08) mm, rotated rx 180 ry 0 rz 180 deg; joints [-140.081, -45.287, -97.416, 46.445, 62.307, -26.049]
  MoveL 9536 to (-19.94, 34.93, 135.08) mm, rotated rx 180 ry 0 rz 180 deg; joints [-140.081, -45.287, -97.416, 46.445, 62.307, -26.049]
  Call Extruder(70.60771)
  MoveL 9537 to (-19.06, 34.91, 135.08) mm, rotated rx -180 ry 0 rz 180 deg; joints [-140.173, -45.333, -97.301, 46.378, 62.219, -26.062]
  Call Extruder(187.25639)
  MoveL 9538 to (219.06, 34.91, 135.08) mm, rotated rx 180 ry 0 rz 180 deg; joints [-155.896, -64.441, -54.991, 42.317, 37.344, -35.899]
  MoveL 9539 to (219.06, 34.91, 135.08) mm, rotated rx 180 ry 0 rz 180 deg; joints [-155.896, -64.441, -54.991, 42.317, 37.344, -35.899]
  Call Extruder(187.97196)
  MoveL 9540 to (220.52, 34.95, 135.08) mm, rotated rx -180 ry 0 rz 180 deg; joints [-155.953, -64.611, -54.639, 42.403, 37.177, -36.04]
  MoveL 9541 to (220.52, 34.95, 135.08) mm, rotated rx -180 ry 0 rz 180 deg; joints [-155.953, -64.611, -54.639, 42.403, 37.177, -36.04]
  Call Extruder(188.54670)
  MoveL 9542 to (221.68, 35, 135.08) mm, rotated rx -180 ry 0 rz -180 deg; joints [-155.997, -64.748, -54.355, 42.475, 37.043, -36.158]
  MoveL 9543 to (221.68, 35, 135.08) mm, rotated rx -180 ry 0 rz -180 deg; joints [-155.997, -64.748, -54.355, 42.475, 37.043, -36.158]
  Call Extruder(188.84009)
  MoveL 9544 to (222.27, 35.04, 135.08) mm, rotated rx -180 ry 0 rz 180 deg; joints [-156.017, -64.82, -54.208, 42.516, 36.975, -36.221]
  MoveL 9545 to (222.27, 35.04, 135.08) mm, rotated rx -180 ry 0 rz 180 deg; joints [-156.017, -64.82, -54.208, 42.516, 36.975, -36.221]
  Call Extruder(189.13482)
  MoveL 9546 to (222.86, 35.09, 135.08) mm, rotated rx 180 ry 0 rz -180 deg; joints [-156.037, -64.891, -54.061, 42.557, 36.908, -36.285]
  MoveL 9547 to (222.86, 35.09, 135.08) mm, rotated rx 180 ry 0 rz -180 deg; joints [-156.037, -64.891, -54.061, 42.557, 36.908, -36.285]
  Call Extruder(189.43087)
  MoveL 9548 to (223.45, 35.14, 135.08) mm, rotated rx 180 ry 0 rz 180 deg; joints [-156.057, -64.963, -53.913, 42.599, 36.84, -36.35]
  MoveL 9549 to (223.45, 35.14, 135.08) mm, rotated rx 180 ry 0 rz 180 deg; joints [-156.057, -64.963, -53.913, 42.599, 36.84, -36.35]
  Call Extruder(189.62715)
  MoveL 9550 to (223.83, 35.18, 135.08) mm, rotated rx -180 ry 0 rz 180 deg; joints [-156.068, -65.01, -53.814, 42.629, 36.795, -36.395]
  MoveL 9551 to (223.83, 35.18, 135.08) mm, rotated rx -180 ry 0 rz 180 deg; joints [-156.068, -65.01, -53.814, 42.629, 36.795, -36.395]
  Call Extruder(189.82429)
  MoveL 9552 to (224.22, 35.23, 135.08) mm, rotated rx -180 ry 0 rz 180 deg; joints [-156.08, -65.059, -53.715, 42.66, 36.751, -36.44]
  MoveL 9553 to (224.22, 35.23, 135.08) mm, rotated rx -180 ry 0 rz 180 deg; joints [-156.08, -65.059, -53.715, 42.66, 36.751, -36.44]
  Call Extruder(190.02230)
  MoveL 9554 to (224.61, 35.27, 135.08) mm, rotated rx -180 ry 0 rz 180 deg; joints [-156.092, -65.107, -53.616, 42.691, 36.707, -36.485]
  MoveL 9555 to (224.61, 35.27, 135.08) mm, rotated rx -180 ry 0 rz 180 deg; joints [-156.092, -65.107, -53.616, 42.691, 36.707, -36.485]
  Call Extruder(190.22117)
  MoveL 9556 to (225, 35.32, 135.08) mm, rotated rx 180 ry 0 rz -180 deg; joints [-156.103, -65.155, -53.517, 42.722, 36.662, -36.531]
  MoveL 9557 to (225, 35.32, 135.08) mm, rotated rx 180 ry 0 rz -180 deg; joints [-156.103, -65.155, -53.517, 42.722, 36.662, -36.531]
  Call Extruder(190.40025)
  MoveL 9558 to (225.34, 35.37, 135.08) mm, rotated rx 180 ry 0 rz 180 deg; joints [-156.113, -65.198, -53.427, 42.751, 36.622, -36.572]
  MoveL 9559 to (225.34, 35.37, 135.08) mm, rotated rx 180 ry 0 rz 180 deg; joints [-156.113, -65.198, -53.427, 42.751, 36.622, -36.572]
  Call Extruder(190.55944)
  MoveL 9560 to (225.65, 35.42, 135.08) mm, rotated rx 180 ry 0 rz 180 deg; joints [-156.121, -65.237, -53.347, 42.777, 36.587, -36.611]
  MoveL 9561 to (225.65, 35.42, 135.08) mm, rotated rx 180 ry 0 rz 180 deg; joints [-156.121, -65.237, -53.347, 42.777, 36.587, -36.611]
  Call Extruder(190.71935)
  MoveL 9562 to (225.96, 35.47, 135.08) mm, rotated rx 180 ry 0 rz 180 deg; joints [-156.129, -65.276, -53.268, 42.804, 36.552, -36.649]
  MoveL 9563 to (225.96, 35.47, 135.08) mm, rotated rx 180 ry 0 rz 180 deg; joints [-156.129, -65.276, -53.268, 42.804, 36.552, -36.649]
  Call Extruder(190.87999)
  MoveL 9564 to (226.26, 35.51, 135.08) mm, rotated rx -180 ry 0 rz 180 deg; joints [-156.137, -65.315, -53.188, 42.831, 36.518, -36.687]
  MoveL 9565 to (226.26, 35.51, 135.08) mm, rotated rx -180 ry 0 rz 180 deg; joints [-156.137, -65.315, -53.188, 42.831, 36.518, -36.687]
  Call Extruder(191.04136)
  MoveL 9566 to (226.57, 35.56, 135.08) mm, rotated rx 180 ry 0 rz 180 deg; joints [-156.145, -65.353, -53.108, 42.858, 36.483, -36.726]
  MoveL 9567 to (226.57, 35.56, 135.08) mm, rotated rx 180 ry 0 rz 180 deg; joints [-156.145, -65.353, -53.108, 42.858, 36.483, -36.726]
  Call Extruder(191.20345)
  MoveL 9568 to (226.87, 35.61, 135.08) mm, rotated rx 180 ry 0 rz -180 deg; joints [-156.153, -65.392, -53.027, 42.886, 36.448, -36.764]
  MoveL 9569 to (226.87, 35.61, 135.08) mm, rotated rx 180 ry 0 rz -180 deg; joints [-156.153, -65.392, -53.027, 42.886, 36.448, -36.764]
  Call Extruder(191.35165)
  MoveL 9570 to (227.15, 35.66, 135.08) mm, rotated rx 180 ry 0 rz 180 deg; joints [-156.16, -65.428, -52.954, 42.911, 36.416, -36.8]
  MoveL 9571 to (227.15, 35.66, 135.08) mm, rotated rx 180 ry 0 rz 180 deg; joints [-156.16, -65.428, -52.954, 42.911, 36.416, -36.8]
  Call Extruder(191.48588)
  MoveL 9572 to (227.4, 35.71, 135.08) mm, rotated rx -180 ry 0 rz 180 deg; joints [-156.165, -65.46, -52.887, 42.935, 36.387, -36.833]
  MoveL 9573 to (227.4, 35.71, 135.08) mm, rotated rx -180 ry 0 rz 180 deg; joints [-156.165, -65.46, -52.887, 42.935, 36.387, -36.833]
  Call Extruder(191.62072)
  MoveL 9574 to (227.65, 35.76, 135.08) mm, rotated rx -180 ry 0 rz 180 deg; joints [-156.171, -65.493, -52.821, 42.96, 36.359, -36.867]
  MoveL 9575 to (227.65, 35.76, 135.08) mm, rotated rx -180 ry 0 rz 180 deg; joints [-156.171, -65.493, -52.821, 42.96, 36.359, -36.867]
  Call Extruder(191.75618)
  MoveL 9576 to (227.9, 35.81, 135.08) mm, rotated rx 180 ry 0 rz 180 deg; joints [-156.176, -65.525, -52.754, 42.984, 36.331, -36.9]
  MoveL 9577 to (227.9, 35.81, 135.08) mm, rotated rx 180 ry 0 rz 180 deg; joints [-156.176, -65.525, -52.754, 42.984, 36.331, -36.9]
  Call Extruder(191.89224)
  MoveL 9578 to (228.15, 35.86, 135.08) mm, rotated rx 180 ry 0 rz 180 deg; joints [-156.182, -65.558, -52.687, 43.008, 36.302, -36.934]
  MoveL 9579 to (228.15, 35.86, 135.08) mm, rotated rx 180 ry 0 rz 180 deg; joints [-156.182, -65.558, -52.687, 43.008, 36.302, -36.934]
  Call Extruder(192.02891)
  MoveL 9580 to (228.4, 35.91, 135.08) mm, rotated rx 180 ry 0 rz 180 deg; joints [-156.187, -65.59, -52.62, 43.033, 36.274, -36.967]
  MoveL 9581 to (228.4, 35.91, 135.08) mm, rotated rx 180 ry 0 rz 180 deg; joints [-156.187, -65.59, -52.62, 43.033, 36.274, -36.967]
  Call Extruder(192.16620)
  MoveL 9582 to (228.65, 35.96, 135.08) mm, rotated rx 180 ry 0 rz 180 deg; joints [-156.193, -65.623, -52.553, 43.057, 36.245, -37.001]
  MoveL 9583 to (228.65, 35.96, 135.08) mm, rotated rx 180 ry 0 rz 180 deg; joints [-156.193, -65.623, -52.553, 43.057, 36.245, -37.001]
  Call Extruder(192.29187)
  MoveL 9584 to (228.87, 36, 135.08) mm, rotated rx -180 ry 0 rz 180 deg; joints [-156.198, -65.652, -52.493, 43.08, 36.219, -37.032]
  MoveL 9585 to (228.87, 36, 135.08) mm, rotated rx -180 ry 0 rz 180 deg; joints [-156.198, -65.652, -52.493, 43.08, 36.219, -37.032]
  Call Extruder(192.40582)
  MoveL 9586 to (229.08, 36.05, 135.08) mm, rotated rx -180 ry 0 rz 180 deg; joints [-156.202, -65.679, -52.437, 43.101, 36.196, -37.06]
  MoveL 9587 to (229.08, 36.05, 135.08) mm, rotated rx -180 ry 0 rz 180 deg; joints [-156.202, -65.679, -52.437, 43.101, 36.196, -37.06]
  Call Extruder(192.52022)
  MoveL 9588 to (229.28, 36.09, 135.08) mm, rotated rx -180 ry 0 rz -180 deg; joints [-156.206, -65.706, -52.382, 43.122, 36.173, -37.089]
  MoveL 9589 to (229.28, 36.09, 135.08) mm, rotated rx -180 ry 0 rz -180 deg; joints [-156.206, -65.706, -52.382, 43.122, 36.173, -37.089]
  Call Extruder(192.63507)
  MoveL 9590 to (229.48, 36.14, 135.08) mm, rotated rx 180 ry 0 rz 180 deg; joints [-156.21, -65.733, -52.326, 43.143, 36.15, -37.117]
  MoveL 9591 to (229.48, 36.14, 135.08) mm, rotated rx 180 ry 0 rz 180 deg; joints [-156.21, -65.733, -52.326, 43.143, 36.15, -37.117]
  Call Extruder(192.75038)
  MoveL 9592 to (229.69, 36.18, 135.08) mm, rotated rx 180 ry 0 rz -180 deg; joints [-156.214, -65.76, -52.271, 43.164, 36.126, -37.146]
  MoveL 9593 to (229.69, 36.18, 135.08) mm, rotated rx 180 ry 0 rz -180 deg; joints [-156.214, -65.76, -52.271, 43.164, 36.126, -37.146]
  Call Extruder(192.82364)
  MoveL 9594 to (229.81, 36.22, 135.08) mm, rotated rx -180 ry 0 rz -180 deg; joints [-156.216, -65.777, -52.235, 43.179, 36.112, -37.165]
  MoveL 9595 to (229.81, 36.22, 135.08) mm, rotated rx -180 ry 0 rz -180 deg; joints [-156.216, -65.777, -52.235, 43.179, 36.112, -37.165]
  Call Extruder(192.95114)
  MoveL 9596 to (230.03, 36.29, 135.08) mm, rotated rx 180 ry 0 rz 180 deg; joints [-156.219, -65.807, -52.173, 43.205, 36.087, -37.199]
  MoveL 9597 to (230.03, 36.29, 135.08) mm, rotated rx 180 ry 0 rz 180 deg; joints [-156.219, -65.807, -52.173, 43.205, 36.087, -37.199]
  Call Extruder(193.07920)
  MoveL 9598 to (230.26, 36.35, 135.08) mm, rotated rx 180 ry 0 rz 180 deg; joints [-156.222, -65.838, -52.111, 43.231, 36.062, -37.233]
  MoveL 9599 to (230.26, 36.35, 135.08) mm, rotated rx 180 ry 0 rz 180 deg; joints [-156.222, -65.838, -52.111, 43.231, 36.062, -37.233]
  Call Extruder(193.20780)
  MoveL 9600 to (230.47, 36.42, 135.08) mm, rotated rx -180 ry 0 rz -180 deg; joints [-156.224, -65.868, -52.049, 43.257, 36.037, -37.267]
  MoveL 9601 to (230.47, 36.42, 135.08) mm, rotated rx -180 ry 0 rz -180 deg; joints [-156.224, -65.868, -52.049, 43.257, 36.037, -37.267]
  Call Extruder(193.33694)
  MoveL 9602 to (230.7, 36.49, 135.08) mm, rotated rx 180 ry 0 rz 180 deg; joints [-156.227, -65.898, -51.987, 43.284, 36.013, -37.301]
  MoveL 9603 to (230.7, 36.49, 135.08) mm, rotated rx 180 ry 0 rz 180 deg; joints [-156.227, -65.898, -51.987, 43.284, 36.013, -37.301]
  Call Extruder(193.44884)
  MoveL 9604 to (230.88, 36.55, 135.08) mm, rotated rx 180 ry 0 rz 180 deg; joints [-156.229, -65.924, -51.934, 43.307, 35.991, -37.331]
  MoveL 9605 to (230.88, 36.55, 135.08) mm, rotated rx 180 ry 0 rz 180 deg; joints [-156.229, -65.924, -51.934, 43.307, 35.991, -37.331]
  Call Extruder(193.56118)
  MoveL 9606 to (231.07, 36.61, 135.08) mm, rotated rx 180 ry 0 rz 180 deg; joints [-156.231, -65.95, -51.88, 43.33, 35.97, -37.361]
  MoveL 9607 to (231.07, 36.61, 135.08) mm, rotated rx 180 ry 0 rz 180 deg; joints [-156.231, -65.95, -51.88, 43.33, 35.97, -37.361]
  Call Extruder(193.67397)
  MoveL 9608 to (231.26, 36.67, 135.08) mm, rotated rx 180 ry 0 rz 180 deg; joints [-156.233, -65.976, -51.826, 43.354, 35.949, -37.391]
  MoveL 9609 to (231.26, 36.67, 135.08) mm, rotated rx 180 ry 0 rz 180 deg; joints [-156.233, -65.976, -51.826, 43.354, 35.949, -37.391]
  Call Extruder(193.78720)
  MoveL 9610 to (231.45, 36.73, 135.08) mm, rotated rx 180 ry 0 rz 180 deg; joints [-156.235, -66.003, -51.772, 43.377, 35.927, -37.421]
  MoveL 9611 to (231.45, 36.73, 135.08) mm, rotated rx 180 ry 0 rz 180 deg; joints [-156.235, -66.003, -51.772, 43.377, 35.927, -37.421]
  Call Extruder(193.90088)
  MoveL 9612 to (231.64, 36.79, 135.08) mm, rotated rx 180 ry 0 rz 180 deg; joints [-156.237, -66.029, -51.719, 43.401, 35.906, -37.451]
  MoveL 9613 to (231.64, 36.79, 135.08) mm, rotated rx 180 ry 0 rz 180 deg; joints [-156.237, -66.029, -51.719, 43.401, 35.906, -37.451]
  Call Extruder(194.08284)
  MoveL 9614 to (231.93, 36.91, 135.08) mm, rotated rx -180 ry 0 rz 180 deg; joints [-156.238, -66.071, -51.632, 43.442, 35.874, -37.502]
  MoveL 9615 to (231.93, 36.91, 135.08) mm, rotated rx -180 ry 0 rz 180 deg; joints [-156.238, -66.071, -51.632, 43.442, 35.874, -37.502]
  Call Extruder(194.26556)
  MoveL 9616 to (232.22, 37.03, 135.08) mm, rotated rx 180 ry 0 rz 180 deg; joints [-156.238, -66.113, -51.546, 43.483, 35.841, -37.554]
  MoveL 9617 to (232.22, 37.03, 135.08) mm, rotated rx 180 ry 0 rz 180 deg; joints [-156.238, -66.113, -51.546, 43.483, 35.841, -37.554]
  Call Extruder(194.43598)
  MoveL 9618 to (232.49, 37.15, 135.08) mm, rotated rx 180 ry 0 rz 180 deg; joints [-156.239, -66.152, -51.466, 43.522, 35.811, -37.602]
  MoveL 9619 to (232.49, 37.15, 135.08) mm, rotated rx 180 ry 0 rz 180 deg; joints [-156.239, -66.152, -51.466, 43.522, 35.811, -37.602]
  Call Extruder(194.59398)
  MoveL 9620 to (232.74, 37.26, 135.08) mm, rotated rx -180 ry 0 rz 180 deg; joints [-156.239, -66.188, -51.391, 43.558, 35.783, -37.646]
  MoveL 9621 to (232.74, 37.26, 135.08) mm, rotated rx -180 ry 0 rz 180 deg; joints [-156.239, -66.188, -51.391, 43.558, 35.783, -37.646]
  Call Extruder(194.75258)
  MoveL 9622 to (232.99, 37.36, 135.08) mm, rotated rx -180 ry 0 rz -180 deg; joints [-156.239, -66.225, -51.317, 43.594, 35.755, -37.691]
  MoveL 9623 to (232.99, 37.36, 135.08) mm, rotated rx -180 ry 0 rz -180 deg; joints [-156.239, -66.225, -51.317, 43.594, 35.755, -37.691]
  Call Extruder(194.95874)
  MoveL 9624 to (233.29, 37.54, 135.08) mm, rotated rx -180 ry 0 rz 180 deg; joints [-156.236, -66.271, -51.221, 43.646, 35.722, -37.753]
  MoveL 9625 to (233.29, 37.54, 135.08) mm, rotated rx -180 ry 0 rz 180 deg; joints [-156.236, -66.271, -51.221, 43.646, 35.722, -37.753]
  Call Extruder(195.16569)
  MoveL 9626 to (233.6, 37.71, 135.08) mm, rotated rx 180 ry 0 rz -180 deg; joints [-156.232, -66.318, -51.125, 43.699, 35.689, -37.816]
  MoveL 9627 to (233.6, 37.71, 135.08) mm, rotated rx 180 ry 0 rz -180 deg; joints [-156.232, -66.318, -51.125, 43.699, 35.689, -37.816]
  Call Extruder(195.37341)
  MoveL 9628 to (233.9, 37.89, 135.08) mm, rotated rx 180 ry 0 rz 180 deg; joints [-156.228, -66.365, -51.029, 43.751, 35.655, -37.878]
  MoveL 9629 to (233.9, 37.89, 135.08) mm, rotated rx 180 ry 0 rz 180 deg; joints [-156.228, -66.365, -51.029, 43.751, 35.655, -37.878]
  Call Extruder(195.58192)
  MoveL 9630 to (234.21, 38.06, 135.08) mm, rotated rx 180 ry 0 rz 180 deg; joints [-156.224, -66.412, -50.932, 43.804, 35.622, -37.941]
  MoveL 9631 to (234.21, 38.06, 135.08) mm, rotated rx 180 ry 0 rz 180 deg; joints [-156.224, -66.412, -50.932, 43.804, 35.622, -37.941]
  Call Extruder(195.76146)
  MoveL 9632 to (234.45, 38.24, 135.08) mm, rotated rx 180 ry 0 rz -180 deg; joints [-156.218, -66.452, -50.851, 43.853, 35.596, -37.997]
  MoveL 9633 to (234.45, 38.24, 135.08) mm, rotated rx 180 ry 0 rz -180 deg; joints [-156.218, -66.452, -50.851, 43.853, 35.596, -37.997]
  Call Extruder(196.09487)
  MoveL 9634 to (234.9, 38.57, 135.08) mm, rotated rx 180 ry 0 rz 180 deg; joints [-156.206, -66.525, -50.7, 43.943, 35.547, -38.102]
  MoveL 9635 to (234.9, 38.57, 135.08) mm, rotated rx 180 ry 0 rz 180 deg; joints [-156.206, -66.525, -50.7, 43.943, 35.547, -38.102]
  Call Extruder(196.42947)
  MoveL 9636 to (235.35, 38.9, 135.08) mm, rotated rx 180 ry 0 rz 180 deg; joints [-156.195, -66.599, -50.549, 44.035, 35.499, -38.208]
  Call Extruder(197.25742)
  MoveL 9637 to (236.39, 39.81, 135.08) mm, rotated rx -180 ry 0 rz 180 deg; joints [-156.154, -66.778, -50.182, 44.274, 35.39, -38.479]
  Call Extruder(198.08537)
  MoveL 9638 to (237.3, 40.85, 135.08) mm, rotated rx -180 ry 0 rz 180 deg; joints [-156.097, -66.95, -49.831, 44.528, 35.297, -38.758]
  Call Extruder(198.25267)
  MoveL 9639 to (237.47, 41.07, 135.08) mm, rotated rx -180 ry 0 rz 180 deg; joints [-156.083, -66.983, -49.763, 44.581, 35.281, -38.816]
  MoveL 9640 to (237.47, 41.07, 135.08) mm, rotated rx -180 ry 0 rz 180 deg; joints [-156.083, -66.983, -49.763, 44.581, 35.281, -38.816]
  Call Extruder(198.58609)
  MoveL 9641 to (237.8, 41.52, 135.08) mm, rotated rx 180 ry 0 rz 180 deg; joints [-156.055, -67.049, -49.628, 44.687, 35.249, -38.93]
  MoveL 9642 to (237.8, 41.52, 135.08) mm, rotated rx 180 ry 0 rz 180 deg; joints [-156.055, -67.049, -49.628, 44.687, 35.249, -38.93]
  Call Extruder(198.91833)
  MoveL 9643 to (238.12, 41.98, 135.08) mm, rotated rx -180 ry 0 rz -180 deg; joints [-156.028, -67.116, -49.491, 44.793, 35.217, -39.046]
  MoveL 9644 to (238.12, 41.98, 135.08) mm, rotated rx -180 ry 0 rz -180 deg; joints [-156.028, -67.116, -49.491, 44.793, 35.217, -39.046]
  Call Extruder(199.03601)
  MoveL 9645 to (238.22, 42.15, 135.08) mm, rotated rx 180 ry 0 rz 180 deg; joints [-156.016, -67.138, -49.446, 44.832, 35.207, -39.086]
  MoveL 9646 to (238.22, 42.15, 135.08) mm, rotated rx 180 ry 0 rz 180 deg; joints [-156.016, -67.138, -49.446, 44.832, 35.207, -39.086]
  Call Extruder(199.24373)
  MoveL 9647 to (238.4, 42.45, 135.08) mm, rotated rx 180 ry 0 rz 180 deg; joints [-155.996, -67.177, -49.366, 44.9, 35.191, -39.159]
  MoveL 9648 to (238.4, 42.45, 135.08) mm, rotated rx 180 ry 0 rz 180 deg; joints [-155.996, -67.177, -49.366, 44.9, 35.191, -39.159]
  Call Extruder(199.45067)
  MoveL 9649 to (238.57, 42.75, 135.08) mm, rotated rx -180 ry 0 rz -180 deg; joints [-155.976, -67.216, -49.286, 44.968, 35.175, -39.231]
  MoveL 9650 to (238.57, 42.75, 135.08) mm, rotated rx -180 ry 0 rz -180 deg; joints [-155.976, -67.216, -49.286, 44.968, 35.175, -39.231]
  Call Extruder(199.65683)
  MoveL 9651 to (238.75, 43.06, 135.08) mm, rotated rx 180 ry 0 rz 180 deg; joints [-155.956, -67.256, -49.205, 45.037, 35.159, -39.304]
  MoveL 9652 to (238.75, 43.06, 135.08) mm, rotated rx 180 ry 0 rz 180 deg; joints [-155.956, -67.256, -49.205, 45.037, 35.159, -39.304]
  Call Extruder(199.83852)
  MoveL 9653 to (238.89, 43.34, 135.08) mm, rotated rx 180 ry 0 rz -180 deg; joints [-155.937, -67.289, -49.137, 45.098, 35.146, -39.368]
  MoveL 9654 to (238.89, 43.34, 135.08) mm, rotated rx 180 ry 0 rz -180 deg; joints [-155.937, -67.289, -49.137, 45.098, 35.146, -39.368]
  Call Extruder(199.99654)
  MoveL 9655 to (239, 43.58, 135.08) mm, rotated rx 180 ry 0 rz -180 deg; joints [-155.919, -67.317, -49.08, 45.151, 35.137, -39.423]
  MoveL 9656 to (239, 43.58, 135.08) mm, rotated rx 180 ry 0 rz -180 deg; joints [-155.919, -67.317, -49.08, 45.151, 35.137, -39.423]
  Call Extruder(200.15395)
  MoveL 9657 to (239.1, 43.83, 135.08) mm, rotated rx 180 ry 0 rz -180 deg; joints [-155.901, -67.344, -49.024, 45.204, 35.128, -39.479]
  MoveL 9658 to (239.1, 43.83, 135.08) mm, rotated rx 180 ry 0 rz -180 deg; joints [-155.901, -67.344, -49.024, 45.204, 35.128, -39.479]
  Call Extruder(200.33666)
  MoveL 9659 to (239.23, 44.12, 135.08) mm, rotated rx 180 ry 0 rz 180 deg; joints [-155.879, -67.376, -48.959, 45.266, 35.118, -39.543]
  MoveL 9660 to (239.23, 44.12, 135.08) mm, rotated rx 180 ry 0 rz 180 deg; joints [-155.879, -67.376, -48.959, 45.266, 35.118, -39.543]
  Call Extruder(200.51862)
  MoveL 9661 to (239.35, 44.42, 135.08) mm, rotated rx 180 ry 0 rz -180 deg; joints [-155.858, -67.408, -48.893, 45.328, 35.109, -39.608]
  MoveL 9662 to (239.35, 44.42, 135.08) mm, rotated rx 180 ry 0 rz -180 deg; joints [-155.858, -67.408, -48.893, 45.328, 35.109, -39.608]
  Call Extruder(200.66595)
  MoveL 9663 to (239.44, 44.66, 135.08) mm, rotated rx 180 ry 0 rz -180 deg; joints [-155.84, -67.434, -48.842, 45.379, 35.101, -39.66]
  MoveL 9664 to (239.44, 44.66, 135.08) mm, rotated rx 180 ry 0 rz -180 deg; joints [-155.84, -67.434, -48.842, 45.379, 35.101, -39.66]
  Call Extruder(200.77919)
  MoveL 9665 to (239.5, 44.85, 135.08) mm, rotated rx 180 ry 0 rz 180 deg; joints [-155.826, -67.452, -48.804, 45.418, 35.097, -39.699]
  MoveL 9666 to (239.5, 44.85, 135.08) mm, rotated rx 180 ry 0 rz 180 deg; joints [-155.826, -67.452, -48.804, 45.418, 35.097, -39.699]
  Call Extruder(200.89198)
  MoveL 9667 to (239.56, 45.03, 135.08) mm, rotated rx -180 ry 0 rz -180 deg; joints [-155.811, -67.471, -48.766, 45.457, 35.093, -39.739]
  MoveL 9668 to (239.56, 45.03, 135.08) mm, rotated rx -180 ry 0 rz -180 deg; joints [-155.811, -67.471, -48.766, 45.457, 35.093, -39.739]
  Call Extruder(201.00432)
  MoveL 9669 to (239.62, 45.22, 135.08) mm, rotated rx -180 ry 0 rz -180 deg; joints [-155.797, -67.489, -48.728, 45.495, 35.088, -39.779]
  MoveL 9670 to (239.62, 45.22, 135.08) mm, rotated rx -180 ry 0 rz -180 deg; joints [-155.797, -67.489, -48.728, 45.495, 35.088, -39.779]
  Call Extruder(201.11622)
  MoveL 9671 to (239.68, 45.41, 135.08) mm, rotated rx -180 ry 0 rz 180 deg; joints [-155.783, -67.508, -48.69, 45.534, 35.084, -39.818]
  MoveL 9672 to (239.68, 45.41, 135.08) mm, rotated rx -180 ry 0 rz 180 deg; joints [-155.783, -67.508, -48.69, 45.534, 35.084, -39.818]
  Call Extruder(201.23762)
  MoveL 9673 to (239.75, 45.62, 135.08) mm, rotated rx 180 ry 0 rz 180 deg; joints [-155.767, -67.528, -48.649, 45.577, 35.079, -39.862]
  MoveL 9674 to (239.75, 45.62, 135.08) mm, rotated rx 180 ry 0 rz 180 deg; joints [-155.767, -67.528, -48.649, 45.577, 35.079, -39.862]
  Call Extruder(201.36842)
  MoveL 9675 to (239.82, 45.84, 135.08) mm, rotated rx 180 ry 0 rz 180 deg; joints [-155.75, -67.549, -48.605, 45.622, 35.075, -39.908]
  MoveL 9676 to (239.82, 45.84, 135.08) mm, rotated rx 180 ry 0 rz 180 deg; joints [-155.75, -67.549, -48.605, 45.622, 35.075, -39.908]
  Call Extruder(201.49864)
  MoveL 9677 to (239.88, 46.06, 135.08) mm, rotated rx 180 ry 0 rz 180 deg; joints [-155.733, -67.571, -48.561, 45.668, 35.07, -39.955]
  MoveL 9678 to (239.88, 46.06, 135.08) mm, rotated rx 180 ry 0 rz 180 deg; joints [-155.733, -67.571, -48.561, 45.668, 35.07, -39.955]
  Call Extruder(201.62830)
  MoveL 9679 to (239.95, 46.29, 135.08) mm, rotated rx -180 ry 0 rz 180 deg; joints [-155.715, -67.592, -48.517, 45.714, 35.065, -40.002]
  MoveL 9680 to (239.95, 46.29, 135.08) mm, rotated rx -180 ry 0 rz 180 deg; joints [-155.715, -67.592, -48.517, 45.714, 35.065, -40.002]
  Call Extruder(201.75740)
  MoveL 9681 to (240.02, 46.51, 135.08) mm, rotated rx -180 ry 0 rz -180 deg; joints [-155.698, -67.614, -48.473, 45.76, 35.061, -40.048]
  MoveL 9682 to (240.02, 46.51, 135.08) mm, rotated rx -180 ry 0 rz -180 deg; joints [-155.698, -67.614, -48.473, 45.76, 35.061, -40.048]
  Call Extruder(201.87246)
  MoveL 9683 to (240.06, 46.72, 135.08) mm, rotated rx 180 ry 0 rz -180 deg; joints [-155.682, -67.631, -48.438, 45.8, 35.059, -40.089]
  MoveL 9684 to (240.06, 46.72, 135.08) mm, rotated rx 180 ry 0 rz -180 deg; joints [-155.682, -67.631, -48.438, 45.8, 35.059, -40.089]
  Call Extruder(201.98706)
  MoveL 9685 to (240.11, 46.92, 135.08) mm, rotated rx 180 ry 0 rz 180 deg; joints [-155.665, -67.649, -48.402, 45.841, 35.057, -40.13]
  MoveL 9686 to (240.11, 46.92, 135.08) mm, rotated rx 180 ry 0 rz 180 deg; joints [-155.665, -67.649, -48.402, 45.841, 35.057, -40.13]
  Call Extruder(202.10121)
  MoveL 9687 to (240.15, 47.12, 135.08) mm, rotated rx 180 ry 0 rz 180 deg; joints [-155.649, -67.666, -48.366, 45.881, 35.054, -40.17]
  MoveL 9688 to (240.15, 47.12, 135.08) mm, rotated rx 180 ry 0 rz 180 deg; joints [-155.649, -67.666, -48.366, 45.881, 35.054, -40.17]
  Call Extruder(202.21491)
  MoveL 9689 to (240.2, 47.33, 135.08) mm, rotated rx 180 ry 0 rz 180 deg; joints [-155.633, -67.684, -48.33, 45.922, 35.052, -40.211]
  MoveL 9690 to (240.2, 47.33, 135.08) mm, rotated rx 180 ry 0 rz 180 deg; joints [-155.633, -67.684, -48.33, 45.922, 35.052, -40.211]
  Call Extruder(202.34032)
  MoveL 9691 to (240.24, 47.55, 135.08) mm, rotated rx -180 ry 0 rz 180 deg; joints [-155.614, -67.703, -48.291, 45.966, 35.05, -40.256]
  MoveL 9692 to (240.24, 47.55, 135.08) mm, rotated rx -180 ry 0 rz 180 deg; joints [-155.614, -67.703, -48.291, 45.966, 35.05, -40.256]
  Call Extruder(202.47730)
  MoveL 9693 to (240.29, 47.8, 135.08) mm, rotated rx -180 ry 0 rz 180 deg; joints [-155.594, -67.724, -48.249, 46.015, 35.048, -40.305]
  MoveL 9694 to (240.29, 47.8, 135.08) mm, rotated rx -180 ry 0 rz 180 deg; joints [-155.594, -67.724, -48.249, 46.015, 35.048, -40.305]
  Call Extruder(202.61366)
  MoveL 9695 to (240.34, 48.05, 135.08) mm, rotated rx -180 ry 0 rz -180 deg; joints [-155.574, -67.745, -48.206, 46.064, 35.046, -40.354]
  MoveL 9696 to (240.34, 48.05, 135.08) mm, rotated rx -180 ry 0 rz -180 deg; joints [-155.574, -67.745, -48.206, 46.064, 35.046, -40.354]
  Call Extruder(202.74942)
  MoveL 9697 to (240.39, 48.3, 135.08) mm, rotated rx 180 ry 0 rz 180 deg; joints [-155.554, -67.766, -48.163, 46.113, 35.044, -40.403]
  MoveL 9698 to (240.39, 48.3, 135.08) mm, rotated rx 180 ry 0 rz 180 deg; joints [-155.554, -67.766, -48.163, 46.113, 35.044, -40.403]
  Call Extruder(202.88457)
  MoveL 9699 to (240.44, 48.55, 135.08) mm, rotated rx 180 ry 0 rz 180 deg; joints [-155.534, -67.787, -48.121, 46.162, 35.042, -40.452]
  MoveL 9700 to (240.44, 48.55, 135.08) mm, rotated rx 180 ry 0 rz 180 deg; joints [-155.534, -67.787, -48.121, 46.162, 35.042, -40.452]
  Call Extruder(203.01910)
  MoveL 9701 to (240.49, 48.8, 135.08) mm, rotated rx 180 ry 0 rz 180 deg; joints [-155.514, -67.808, -48.078, 46.211, 35.04, -40.501]
  MoveL 9702 to (240.49, 48.8, 135.08) mm, rotated rx 180 ry 0 rz 180 deg; joints [-155.514, -67.808, -48.078, 46.211, 35.04, -40.501]
  Call Extruder(203.15303)
  MoveL 9703 to (240.54, 49.05, 135.08) mm, rotated rx 180 ry 0 rz 180 deg; joints [-155.494, -67.829, -48.035, 46.26, 35.038, -40.55]
  MoveL 9704 to (240.54, 49.05, 135.08) mm, rotated rx 180 ry 0 rz 180 deg; joints [-155.494, -67.829, -48.035, 46.26, 35.038, -40.55]
  Call Extruder(203.30090)
  MoveL 9705 to (240.59, 49.33, 135.08) mm, rotated rx -180 ry 0 rz -180 deg; joints [-155.471, -67.851, -47.99, 46.314, 35.037, -40.604]
  MoveL 9706 to (240.59, 49.33, 135.08) mm, rotated rx -180 ry 0 rz -180 deg; joints [-155.471, -67.851, -47.99, 46.314, 35.037, -40.604]
  Call Extruder(203.46264)
  MoveL 9707 to (240.64, 49.63, 135.08) mm, rotated rx -180 ry 0 rz -180 deg; joints [-155.446, -67.875, -47.94, 46.373, 35.035, -40.663]
  MoveL 9708 to (240.64, 49.63, 135.08) mm, rotated rx -180 ry 0 rz -180 deg; joints [-155.446, -67.875, -47.94, 46.373, 35.035, -40.663]
  Call Extruder(203.62365)
  MoveL 9709 to (240.69, 49.94, 135.08) mm, rotated rx 180 ry 0 rz -180 deg; joints [-155.421, -67.9, -47.891, 46.433, 35.035, -40.722]
  MoveL 9710 to (240.69, 49.94, 135.08) mm, rotated rx 180 ry 0 rz -180 deg; joints [-155.421, -67.9, -47.891, 46.433, 35.035, -40.722]
  Call Extruder(203.78394)
  MoveL 9711 to (240.74, 50.24, 135.08) mm, rotated rx -180 ry 0 rz 180 deg; joints [-155.396, -67.924, -47.841, 46.492, 35.033, -40.781]
  MoveL 9712 to (240.74, 50.24, 135.08) mm, rotated rx -180 ry 0 rz 180 deg; joints [-155.396, -67.924, -47.841, 46.492, 35.033, -40.781]
  Call Extruder(203.94350)
  MoveL 9713 to (240.78, 50.55, 135.08) mm, rotated rx 180 ry 0 rz 180 deg; joints [-155.371, -67.948, -47.792, 46.551, 35.033, -40.84]
  MoveL 9714 to (240.78, 50.55, 135.08) mm, rotated rx 180 ry 0 rz 180 deg; joints [-155.371, -67.948, -47.792, 46.551, 35.033, -40.84]
  Call Extruder(204.10233)
  MoveL 9715 to (240.83, 50.86, 135.08) mm, rotated rx -180 ry 0 rz 180 deg; joints [-155.346, -67.973, -47.742, 46.61, 35.031, -40.899]
  MoveL 9716 to (240.83, 50.86, 135.08) mm, rotated rx -180 ry 0 rz 180 deg; joints [-155.346, -67.973, -47.742, 46.61, 35.031, -40.899]
  Call Extruder(204.28100)
  MoveL 9717 to (240.88, 51.2, 135.08) mm, rotated rx 180 ry 0 rz 180 deg; joints [-155.317, -67.999, -47.688, 46.676, 35.031, -40.965]
  MoveL 9718 to (240.88, 51.2, 135.08) mm, rotated rx 180 ry 0 rz 180 deg; joints [-155.317, -67.999, -47.688, 46.676, 35.031, -40.965]
  Call Extruder(204.47945)
  MoveL 9719 to (240.92, 51.59, 135.08) mm, rotated rx 180 ry 0 rz -180 deg; joints [-155.285, -68.028, -47.629, 46.75, 35.032, -41.038]
  MoveL 9720 to (240.92, 51.59, 135.08) mm, rotated rx 180 ry 0 rz -180 deg; joints [-155.285, -68.028, -47.629, 46.75, 35.032, -41.038]
  Call Extruder(204.67702)
  MoveL 9721 to (240.97, 51.98, 135.08) mm, rotated rx 180 ry 0 rz 180 deg; joints [-155.252, -68.057, -47.57, 46.824, 35.033, -41.111]
  MoveL 9722 to (240.97, 51.98, 135.08) mm, rotated rx 180 ry 0 rz 180 deg; joints [-155.252, -68.057, -47.57, 46.824, 35.033, -41.111]
  Call Extruder(204.87373)
  MoveL 9723 to (241.02, 52.36, 135.08) mm, rotated rx -180 ry 0 rz 180 deg; joints [-155.22, -68.086, -47.51, 46.898, 35.033, -41.184]
  MoveL 9724 to (241.02, 52.36, 135.08) mm, rotated rx -180 ry 0 rz 180 deg; joints [-155.22, -68.086, -47.51, 46.898, 35.033, -41.184]
  Call Extruder(205.06957)
  MoveL 9725 to (241.06, 52.75, 135.08) mm, rotated rx 180 ry 0 rz 180 deg; joints [-155.188, -68.115, -47.451, 46.971, 35.034, -41.257]
  MoveL 9726 to (241.06, 52.75, 135.08) mm, rotated rx 180 ry 0 rz 180 deg; joints [-155.188, -68.115, -47.451, 46.971, 35.034, -41.257]
  Call Extruder(205.36500)
  MoveL 9727 to (241.11, 53.34, 135.08) mm, rotated rx -180 ry 0 rz 180 deg; joints [-155.138, -68.157, -47.367, 47.082, 35.038, -41.365]
  MoveL 9728 to (241.11, 53.34, 135.08) mm, rotated rx -180 ry 0 rz 180 deg; joints [-155.138, -68.157, -47.367, 47.082, 35.038, -41.365]
  Call Extruder(205.65911)
  MoveL 9729 to (241.16, 53.93, 135.08) mm, rotated rx 180 ry 0 rz 180 deg; joints [-155.088, -68.198, -47.282, 47.192, 35.041, -41.474]
  MoveL 9730 to (241.16, 53.93, 135.08) mm, rotated rx 180 ry 0 rz 180 deg; joints [-155.088, -68.198, -47.282, 47.192, 35.041, -41.474]
  Call Extruder(205.95189)
  MoveL 9731 to (241.2, 54.52, 135.08) mm, rotated rx -180 ry 0 rz -180 deg; joints [-155.038, -68.24, -47.197, 47.302, 35.045, -41.582]
  MoveL 9732 to (241.2, 54.52, 135.08) mm, rotated rx -180 ry 0 rz -180 deg; joints [-155.038, -68.24, -47.197, 47.302, 35.045, -41.582]
  Call Extruder(206.52534)
  MoveL 9733 to (241.25, 55.68, 135.08) mm, rotated rx 180 ry 0 rz 180 deg; joints [-154.938, -68.316, -47.042, 47.516, 35.058, -41.79]
  MoveL 9734 to (241.25, 55.68, 135.08) mm, rotated rx 180 ry 0 rz 180 deg; joints [-154.938, -68.316, -47.042, 47.516, 35.058, -41.79]
  Call Extruder(207.23917)
  MoveL 9735 to (241.29, 57.14, 135.08) mm, rotated rx -180 ry 0 rz 180 deg; joints [-154.812, -68.41, -46.85, 47.781, 35.077, -42.049]
  Call Extruder(249.30405)
  MoveL 9736 to (241.29, 142.86, 135.08) mm, rotated rx 180 ry 0 rz 180 deg; joints [-147.778, -75.141, -33.305, 63.342, 36.628, -57.972]
  Call Extruder(249.73248)
  MoveL 9737 to (241.27, 143.73, 135.08) mm, rotated rx -180 ry 0 rz 180 deg; joints [-147.711, -75.225, -33.136, 63.503, 36.648, -58.146]
  MoveL 9738 to (241.27, 143.73, 135.08) mm, rotated rx -180 ry 0 rz 180 deg; joints [-147.711, -75.225, -33.136, 63.503, 36.648, -58.146]
  Call Extruder(250.30594)
  MoveL 9739 to (241.23, 144.9, 135.08) mm, rotated rx 180 ry 0 rz 180 deg; joints [-147.62, -75.336, -32.917, 63.715, 36.676, -58.374]
  MoveL 9740 to (241.23, 144.9, 135.08) mm, rotated rx 180 ry 0 rz 180 deg; joints [-147.62, -75.336, -32.917, 63.715, 36.676, -58.374]
  Call Extruder(250.74027)
  MoveL 9741 to (241.18, 145.77, 135.08) mm, rotated rx -180 ry 0 rz 180 deg; joints [-147.551, -75.417, -32.754, 63.873, 36.699, -58.544]
  MoveL 9742 to (241.18, 145.77, 135.08) mm, rotated rx -180 ry 0 rz 180 deg; joints [-147.551, -75.417, -32.754, 63.873, 36.699, -58.544]
  Call Extruder(251.03438)
  MoveL 9743 to (241.13, 146.36, 135.08) mm, rotated rx -180 ry 0 rz -180 deg; joints [-147.504, -75.47, -32.649, 63.977, 36.717, -58.655]
  MoveL 9744 to (241.13, 146.36, 135.08) mm, rotated rx -180 ry 0 rz -180 deg; joints [-147.504, -75.47, -32.649, 63.977, 36.717, -58.655]
  Call Extruder(251.32982)
  MoveL 9745 to (241.09, 146.95, 135.08) mm, rotated rx 180 ry 0 rz -180 deg; joints [-147.457, -75.523, -32.544, 64.081, 36.734, -58.767]
  MoveL 9746 to (241.09, 146.95, 135.08) mm, rotated rx 180 ry 0 rz -180 deg; joints [-147.457, -75.523, -32.544, 64.081, 36.734, -58.767]
  Call Extruder(251.57607)
  MoveL 9747 to (241.04, 147.44, 135.08) mm, rotated rx -180 ry 0 rz 180 deg; joints [-147.417, -75.566, -32.459, 64.166, 36.749, -58.858]
  MoveL 9748 to (241.04, 147.44, 135.08) mm, rotated rx -180 ry 0 rz 180 deg; joints [-147.417, -75.566, -32.459, 64.166, 36.749, -58.858]
  Call Extruder(251.77278)
  MoveL 9749 to (240.99, 147.83, 135.08) mm, rotated rx -180 ry 0 rz 180 deg; joints [-147.386, -75.598, -32.394, 64.232, 36.762, -58.928]
  MoveL 9750 to (240.99, 147.83, 135.08) mm, rotated rx -180 ry 0 rz 180 deg; joints [-147.386, -75.598, -32.394, 64.232, 36.762, -58.928]
  Call Extruder(251.97035)
  MoveL 9751 to (240.95, 148.22, 135.08) mm, rotated rx -180 ry 0 rz 180 deg; joints [-147.354, -75.631, -32.329, 64.298, 36.775, -58.999]
  MoveL 9752 to (240.95, 148.22, 135.08) mm, rotated rx -180 ry 0 rz 180 deg; joints [-147.354, -75.631, -32.329, 64.298, 36.775, -58.999]
  Call Extruder(252.16879)
  MoveL 9753 to (240.9, 148.6, 135.08) mm, rotated rx 180 ry 0 rz -180 deg; joints [-147.322, -75.664, -32.264, 64.364, 36.788, -59.069]
  MoveL 9754 to (240.9, 148.6, 135.08) mm, rotated rx 180 ry 0 rz -180 deg; joints [-147.322, -75.664, -32.264, 64.364, 36.788, -59.069]
  Call Extruder(252.36810)
  MoveL 9755 to (240.86, 148.99, 135.08) mm, rotated rx 180 ry 0 rz 180 deg; joints [-147.291, -75.696, -32.199, 64.43, 36.802, -59.14]
  MoveL 9756 to (240.86, 148.99, 135.08) mm, rotated rx 180 ry 0 rz 180 deg; joints [-147.291, -75.696, -32.199, 64.43, 36.802, -59.14]
  Call Extruder(252.52693)
  MoveL 9757 to (240.81, 149.3, 135.08) mm, rotated rx -180 ry 0 rz 180 deg; joints [-147.265, -75.72, -32.151, 64.481, 36.813, -59.193]
  MoveL 9758 to (240.81, 149.3, 135.08) mm, rotated rx -180 ry 0 rz 180 deg; joints [-147.265, -75.72, -32.151, 64.481, 36.813, -59.193]
  Call Extruder(252.68649)
  MoveL 9759 to (240.76, 149.6, 135.08) mm, rotated rx 180 ry 0 rz -180 deg; joints [-147.24, -75.744, -32.103, 64.531, 36.825, -59.246]
  MoveL 9760 to (240.76, 149.6, 135.08) mm, rotated rx 180 ry 0 rz -180 deg; joints [-147.24, -75.744, -32.103, 64.531, 36.825, -59.246]
  Call Extruder(252.84678)
  MoveL 9761 to (240.71, 149.91, 135.08) mm, rotated rx 180 ry 0 rz 180 deg; joints [-147.214, -75.768, -32.056, 64.582, 36.837, -59.299]
  MoveL 9762 to (240.71, 149.91, 135.08) mm, rotated rx 180 ry 0 rz 180 deg; joints [-147.214, -75.768, -32.056, 64.582, 36.837, -59.299]
  Call Extruder(253.00780)
  MoveL 9763 to (240.66, 150.21, 135.08) mm, rotated rx -180 ry 0 rz -180 deg; joints [-147.189, -75.793, -32.008, 64.632, 36.848, -59.352]
  MoveL 9764 to (240.66, 150.21, 135.08) mm, rotated rx -180 ry 0 rz -180 deg; joints [-147.189, -75.793, -32.008, 64.632, 36.848, -59.352]
  Call Extruder(253.16954)
  MoveL 9765 to (240.61, 150.52, 135.08) mm, rotated rx 180 ry 0 rz 180 deg; joints [-147.163, -75.817, -31.96, 64.683, 36.86, -59.406]
  MoveL 9766 to (240.61, 150.52, 135.08) mm, rotated rx 180 ry 0 rz 180 deg; joints [-147.163, -75.817, -31.96, 64.683, 36.86, -59.406]
  Call Extruder(253.33202)
  MoveL 9767 to (240.56, 150.83, 135.08) mm, rotated rx 180 ry 0 rz -180 deg; joints [-147.138, -75.841, -31.912, 64.733, 36.872, -59.459]
  MoveL 9768 to (240.56, 150.83, 135.08) mm, rotated rx 180 ry 0 rz -180 deg; joints [-147.138, -75.841, -31.912, 64.733, 36.872, -59.459]
  Call Extruder(253.46594)
  MoveL 9769 to (240.52, 151.07, 135.08) mm, rotated rx 180 ry 0 rz 180 deg; joints [-147.117, -75.859, -31.875, 64.773, 36.882, -59.501]
  MoveL 9770 to (240.52, 151.07, 135.08) mm, rotated rx 180 ry 0 rz 180 deg; joints [-147.117, -75.859, -31.875, 64.773, 36.882, -59.501]
  Call Extruder(253.60048)
  MoveL 9771 to (240.47, 151.32, 135.08) mm, rotated rx -180 ry 0 rz -180 deg; joints [-147.095, -75.877, -31.839, 64.812, 36.893, -59.542]
  MoveL 9772 to (240.47, 151.32, 135.08) mm, rotated rx -180 ry 0 rz -180 deg; joints [-147.095, -75.877, -31.839, 64.812, 36.893, -59.542]
  Call Extruder(253.73563)
  MoveL 9773 to (240.42, 151.57, 135.08) mm, rotated rx 180 ry 0 rz 180 deg; joints [-147.074, -75.895, -31.803, 64.852, 36.904, -59.583]
  MoveL 9774 to (240.42, 151.57, 135.08) mm, rotated rx 180 ry 0 rz 180 deg; joints [-147.074, -75.895, -31.803, 64.852, 36.904, -59.583]
  Call Extruder(253.87138)
  MoveL 9775 to (240.37, 151.82, 135.08) mm, rotated rx -180 ry 0 rz -180 deg; joints [-147.053, -75.914, -31.767, 64.891, 36.914, -59.625]
  MoveL 9776 to (240.37, 151.82, 135.08) mm, rotated rx -180 ry 0 rz -180 deg; joints [-147.053, -75.914, -31.767, 64.891, 36.914, -59.625]
  Call Extruder(254.00775)
  MoveL 9777 to (240.32, 152.07, 135.08) mm, rotated rx 180 ry 0 rz 180 deg; joints [-147.032, -75.932, -31.731, 64.931, 36.925, -59.666]
  MoveL 9778 to (240.32, 152.07, 135.08) mm, rotated rx 180 ry 0 rz 180 deg; joints [-147.032, -75.932, -31.731, 64.931, 36.925, -59.666]
  Call Extruder(254.14473)
  MoveL 9779 to (240.27, 152.32, 135.08) mm, rotated rx -180 ry 0 rz -180 deg; joints [-147.011, -75.95, -31.694, 64.97, 36.936, -59.707]
  MoveL 9780 to (240.27, 152.32, 135.08) mm, rotated rx -180 ry 0 rz -180 deg; joints [-147.011, -75.95, -31.694, 64.97, 36.936, -59.707]
  Call Extruder(254.28232)
  MoveL 9781 to (240.22, 152.57, 135.08) mm, rotated rx 180 ry 0 rz -180 deg; joints [-146.989, -75.968, -31.658, 65.01, 36.946, -59.749]
  MoveL 9782 to (240.22, 152.57, 135.08) mm, rotated rx 180 ry 0 rz -180 deg; joints [-146.989, -75.968, -31.658, 65.01, 36.946, -59.749]
  Call Extruder(254.39601)
  MoveL 9783 to (240.17, 152.77, 135.08) mm, rotated rx 180 ry 0 rz 180 deg; joints [-146.972, -75.983, -31.629, 65.042, 36.956, -59.782]
  MoveL 9784 to (240.17, 152.77, 135.08) mm, rotated rx 180 ry 0 rz 180 deg; joints [-146.972, -75.983, -31.629, 65.042, 36.956, -59.782]
  Call Extruder(254.51016)
  MoveL 9785 to (240.13, 152.98, 135.08) mm, rotated rx 180 ry 0 rz -180 deg; joints [-146.954, -75.997, -31.601, 65.074, 36.965, -59.815]
  MoveL 9786 to (240.13, 152.98, 135.08) mm, rotated rx 180 ry 0 rz -180 deg; joints [-146.954, -75.997, -31.601, 65.074, 36.965, -59.815]
  Call Extruder(254.62477)
  MoveL 9787 to (240.08, 153.18, 135.08) mm, rotated rx -180 ry 0 rz 180 deg; joints [-146.937, -76.012, -31.572, 65.105, 36.974, -59.848]
  MoveL 9788 to (240.08, 153.18, 135.08) mm, rotated rx -180 ry 0 rz 180 deg; joints [-146.937, -76.012, -31.572, 65.105, 36.974, -59.848]
  Call Extruder(254.73982)
  MoveL 9789 to (240.04, 153.39, 135.08) mm, rotated rx -180 ry 0 rz -180 deg; joints [-146.919, -76.026, -31.543, 65.137, 36.983, -59.882]
  MoveL 9790 to (240.04, 153.39, 135.08) mm, rotated rx -180 ry 0 rz -180 deg; joints [-146.919, -76.026, -31.543, 65.137, 36.983, -59.882]
  Call Extruder(254.86204)
  MoveL 9791 to (239.98, 153.6, 135.08) mm, rotated rx 180 ry 0 rz -180 deg; joints [-146.9, -76.04, -31.516, 65.169, 36.994, -59.915]
  MoveL 9792 to (239.98, 153.6, 135.08) mm, rotated rx 180 ry 0 rz -180 deg; joints [-146.9, -76.04, -31.516, 65.169, 36.994, -59.915]
  Call Extruder(254.99170)
  MoveL 9793 to (239.92, 153.82, 135.08) mm, rotated rx 180 ry 0 rz -180 deg; joints [-146.88, -76.053, -31.491, 65.201, 37.006, -59.947]
  MoveL 9794 to (239.92, 153.82, 135.08) mm, rotated rx 180 ry 0 rz -180 deg; joints [-146.88, -76.053, -31.491, 65.201, 37.006, -59.947]
  Call Extruder(255.12193)
  MoveL 9795 to (239.85, 154.05, 135.08) mm, rotated rx 180 ry 0 rz 180 deg; joints [-146.86, -76.065, -31.466, 65.233, 37.018, -59.979]
  MoveL 9796 to (239.85, 154.05, 135.08) mm, rotated rx 180 ry 0 rz 180 deg; joints [-146.86, -76.065, -31.466, 65.233, 37.018, -59.979]
  Call Extruder(255.25272)
  MoveL 9797 to (239.78, 154.27, 135.08) mm, rotated rx 180 ry 0 rz -180 deg; joints [-146.84, -76.078, -31.44, 65.265, 37.03, -60.012]
  MoveL 9798 to (239.78, 154.27, 135.08) mm, rotated rx 180 ry 0 rz -180 deg; joints [-146.84, -76.078, -31.44, 65.265, 37.03, -60.012]
  Call Extruder(255.38407)
  MoveL 9799 to (239.71, 154.49, 135.08) mm, rotated rx -180 ry 0 rz -180 deg; joints [-146.82, -76.091, -31.414, 65.297, 37.042, -60.044]
  MoveL 9800 to (239.71, 154.49, 135.08) mm, rotated rx -180 ry 0 rz -180 deg; joints [-146.82, -76.091, -31.414, 65.297, 37.042, -60.044]
  Call Extruder(255.49598)
  MoveL 9801 to (239.65, 154.68, 135.08) mm, rotated rx -180 ry 0 rz -180 deg; joints [-146.803, -76.101, -31.394, 65.323, 37.053, -60.071]
  MoveL 9802 to (239.65, 154.68, 135.08) mm, rotated rx -180 ry 0 rz -180 deg; joints [-146.803, -76.101, -31.394, 65.323, 37.053, -60.071]
  Call Extruder(255.60832)
  MoveL 9803 to (239.59, 154.87, 135.08) mm, rotated rx -180 ry 0 rz 180 deg; joints [-146.785, -76.112, -31.374, 65.35, 37.064, -60.097]
  MoveL 9804 to (239.59, 154.87, 135.08) mm, rotated rx -180 ry 0 rz 180 deg; joints [-146.785, -76.112, -31.374, 65.35, 37.064, -60.097]
  Call Extruder(255.72111)
  MoveL 9805 to (239.53, 155.06, 135.08) mm, rotated rx -180 ry 0 rz 180 deg; joints [-146.768, -76.122, -31.354, 65.376, 37.074, -60.124]
  MoveL 9806 to (239.53, 155.06, 135.08) mm, rotated rx -180 ry 0 rz 180 deg; joints [-146.768, -76.122, -31.354, 65.376, 37.074, -60.124]
  Call Extruder(255.83435)
  MoveL 9807 to (239.47, 155.25, 135.08) mm, rotated rx 180 ry 0 rz 180 deg; joints [-146.751, -76.132, -31.333, 65.402, 37.085, -60.15]
  MoveL 9808 to (239.47, 155.25, 135.08) mm, rotated rx 180 ry 0 rz 180 deg; joints [-146.751, -76.132, -31.333, 65.402, 37.085, -60.15]
  Call Extruder(255.94803)
  MoveL 9809 to (239.41, 155.44, 135.08) mm, rotated rx 180 ry 0 rz 180 deg; joints [-146.734, -76.142, -31.313, 65.428, 37.096, -60.177]
  MoveL 9810 to (239.41, 155.44, 135.08) mm, rotated rx 180 ry 0 rz 180 deg; joints [-146.734, -76.142, -31.313, 65.428, 37.096, -60.177]
  Call Extruder(256.12998)
  MoveL 9811 to (239.29, 155.73, 135.08) mm, rotated rx 180 ry 0 rz -180 deg; joints [-146.706, -76.154, -31.29, 65.465, 37.115, -60.212]
  MoveL 9812 to (239.29, 155.73, 135.08) mm, rotated rx 180 ry 0 rz -180 deg; joints [-146.706, -76.154, -31.29, 65.465, 37.115, -60.212]
  Call Extruder(256.31270)
  MoveL 9813 to (239.16, 156.02, 135.08) mm, rotated rx 180 ry 0 rz 180 deg; joints [-146.678, -76.165, -31.267, 65.502, 37.134, -60.248]
  MoveL 9814 to (239.16, 156.02, 135.08) mm, rotated rx 180 ry 0 rz 180 deg; joints [-146.678, -76.165, -31.267, 65.502, 37.134, -60.248]
  Call Extruder(256.48312)
  MoveL 9815 to (239.05, 156.29, 135.08) mm, rotated rx -180 ry 0 rz -180 deg; joints [-146.652, -76.176, -31.246, 65.535, 37.153, -60.28]
  MoveL 9816 to (239.05, 156.29, 135.08) mm, rotated rx -180 ry 0 rz -180 deg; joints [-146.652, -76.176, -31.246, 65.535, 37.153, -60.28]
  Call Extruder(256.64113)
  MoveL 9817 to (238.94, 156.54, 135.08) mm, rotated rx 180 ry 0 rz 180 deg; joints [-146.628, -76.185, -31.228, 65.566, 37.17, -60.31]
  MoveL 9818 to (238.94, 156.54, 135.08) mm, rotated rx 180 ry 0 rz 180 deg; joints [-146.628, -76.185, -31.228, 65.566, 37.17, -60.31]
  Call Extruder(256.79975)
  MoveL 9819 to (238.84, 156.79, 135.08) mm, rotated rx -180 ry 0 rz 180 deg; joints [-146.604, -76.195, -31.209, 65.597, 37.187, -60.34]
  MoveL 9820 to (238.84, 156.79, 135.08) mm, rotated rx -180 ry 0 rz 180 deg; joints [-146.604, -76.195, -31.209, 65.597, 37.187, -60.34]
  Call Extruder(257.00592)
  MoveL 9821 to (238.66, 157.09, 135.08) mm, rotated rx -180 ry 0 rz 180 deg; joints [-146.573, -76.199, -31.2, 65.628, 37.212, -60.366]
  MoveL 9822 to (238.66, 157.09, 135.08) mm, rotated rx -180 ry 0 rz 180 deg; joints [-146.573, -76.199, -31.2, 65.628, 37.212, -60.366]
  Call Extruder(257.21287)
  MoveL 9823 to (238.49, 157.4, 135.08) mm, rotated rx -180 ry 0 rz 180 deg; joints [-146.542, -76.203, -31.192, 65.658, 37.238, -60.393]
  MoveL 9824 to (238.49, 157.4, 135.08) mm, rotated rx -180 ry 0 rz 180 deg; joints [-146.542, -76.203, -31.192, 65.658, 37.238, -60.393]
  Call Extruder(257.42059)
  MoveL 9825 to (238.31, 157.7, 135.08) mm, rotated rx -180 ry 0 rz -180 deg; joints [-146.51, -76.207, -31.184, 65.689, 37.263, -60.42]
  MoveL 9826 to (238.31, 157.7, 135.08) mm, rotated rx -180 ry 0 rz -180 deg; joints [-146.51, -76.207, -31.184, 65.689, 37.263, -60.42]
  Call Extruder(257.62910)
  MoveL 9827 to (238.13, 158.01, 135.08) mm, rotated rx 180 ry 0 rz -180 deg; joints [-146.479, -76.211, -31.176, 65.719, 37.289, -60.446]
  MoveL 9828 to (238.13, 158.01, 135.08) mm, rotated rx 180 ry 0 rz -180 deg; joints [-146.479, -76.211, -31.176, 65.719, 37.289, -60.446]
  Call Extruder(257.80864)
  MoveL 9829 to (237.96, 158.25, 135.08) mm, rotated rx -180 ry 0 rz 180 deg; joints [-146.452, -76.209, -31.18, 65.739, 37.313, -60.46]
  MoveL 9830 to (237.96, 158.25, 135.08) mm, rotated rx -180 ry 0 rz 180 deg; joints [-146.452, -76.209, -31.18, 65.739, 37.313, -60.46]
  Call Extruder(258.14205)
  MoveL 9831 to (237.63, 158.7, 135.08) mm, rotated rx 180 ry 0 rz 180 deg; joints [-146.402, -76.204, -31.189, 65.774, 37.359, -60.486]
  MoveL 9832 to (237.63, 158.7, 135.08) mm, rotated rx 180 ry 0 rz 180 deg; joints [-146.402, -76.204, -31.189, 65.774, 37.359, -60.486]
  Call Extruder(258.47664)
  MoveL 9833 to (237.3, 159.15, 135.08) mm, rotated rx 180 ry 0 rz 180 deg; joints [-146.352, -76.2, -31.198, 65.809, 37.404, -60.511]
  Call Extruder(259.30463)
  MoveL 9834 to (236.39, 160.19, 135.08) mm, rotated rx 180 ry 0 rz 180 deg; joints [-146.229, -76.164, -31.27, 65.866, 37.526, -60.537]
  Call Extruder(260.13252)
  MoveL 9835 to (235.35, 161.1, 135.08) mm, rotated rx -180 ry 0 rz -180 deg; joints [-146.109, -76.095, -31.408, 65.882, 37.658, -60.511]
  Call Extruder(260.29983)
  MoveL 9836 to (235.13, 161.27, 135.08) mm, rotated rx -180 ry 0 rz -180 deg; joints [-146.086, -76.076, -31.445, 65.879, 37.686, -60.498]
  MoveL 9837 to (235.13, 161.27, 135.08) mm, rotated rx -180 ry 0 rz -180 deg; joints [-146.086, -76.076, -31.445, 65.879, 37.686, -60.498]
  Call Extruder(260.63326)
  MoveL 9838 to (234.68, 161.59, 135.08) mm, rotated rx 180 ry 0 rz 180 deg; joints [-146.039, -76.038, -31.519, 65.873, 37.742, -60.473]
  MoveL 9839 to (234.68, 161.59, 135.08) mm, rotated rx 180 ry 0 rz 180 deg; joints [-146.039, -76.038, -31.519, 65.873, 37.742, -60.473]
  Call Extruder(260.96550)
  MoveL 9840 to (234.22, 161.92, 135.08) mm, rotated rx -180 ry 0 rz 180 deg; joints [-145.992, -76.001, -31.593, 65.868, 37.798, -60.448]
  MoveL 9841 to (234.22, 161.92, 135.08) mm, rotated rx -180 ry 0 rz 180 deg; joints [-145.992, -76.001, -31.593, 65.868, 37.798, -60.448]
  Call Extruder(261.08316)
  MoveL 9842 to (234.05, 162.02, 135.08) mm, rotated rx 180 ry 0 rz 180 deg; joints [-145.976, -75.984, -31.627, 65.861, 37.819, -60.434]
  MoveL 9843 to (234.05, 162.02, 135.08) mm, rotated rx 180 ry 0 rz 180 deg; joints [-145.976, -75.984, -31.627, 65.861, 37.819, -60.434]
  Call Extruder(261.29090)
  MoveL 9844 to (233.75, 162.2, 135.08) mm, rotated rx 180 ry 0 rz 180 deg; joints [-145.947, -75.954, -31.686, 65.849, 37.855, -60.408]
  MoveL 9845 to (233.75, 162.2, 135.08) mm, rotated rx 180 ry 0 rz 180 deg; joints [-145.947, -75.954, -31.686, 65.849, 37.855, -60.408]
  Call Extruder(261.49785)
  MoveL 9846 to (233.45, 162.37, 135.08) mm, rotated rx -180 ry 0 rz 180 deg; joints [-145.919, -75.924, -31.745, 65.837, 37.892, -60.382]
  MoveL 9847 to (233.45, 162.37, 135.08) mm, rotated rx -180 ry 0 rz 180 deg; joints [-145.919, -75.924, -31.745, 65.837, 37.892, -60.382]
  Call Extruder(261.70402)
  MoveL 9848 to (233.14, 162.55, 135.08) mm, rotated rx 180 ry 0 rz -180 deg; joints [-145.891, -75.895, -31.805, 65.826, 37.929, -60.356]
  MoveL 9849 to (233.14, 162.55, 135.08) mm, rotated rx 180 ry 0 rz -180 deg; joints [-145.891, -75.895, -31.805, 65.826, 37.929, -60.356]
  Call Extruder(261.88569)
  MoveL 9850 to (232.86, 162.69, 135.08) mm, rotated rx 180 ry 0 rz 180 deg; joints [-145.866, -75.866, -31.862, 65.812, 37.962, -60.329]
  MoveL 9851 to (232.86, 162.69, 135.08) mm, rotated rx 180 ry 0 rz 180 deg; joints [-145.866, -75.866, -31.862, 65.812, 37.962, -60.329]
  Call Extruder(262.04366)
  MoveL 9852 to (232.62, 162.8, 135.08) mm, rotated rx -180 ry 0 rz -180 deg; joints [-145.845, -75.837, -31.919, 65.796, 37.991, -60.301]
  MoveL 9853 to (232.62, 162.8, 135.08) mm, rotated rx -180 ry 0 rz -180 deg; joints [-145.845, -75.837, -31.919, 65.796, 37.991, -60.301]
  Call Extruder(262.20102)
  MoveL 9854 to (232.37, 162.91, 135.08) mm, rotated rx -180 ry 0 rz 180 deg; joints [-145.825, -75.809, -31.975, 65.78, 38.02, -60.273]
  MoveL 9855 to (232.37, 162.91, 135.08) mm, rotated rx -180 ry 0 rz 180 deg; joints [-145.825, -75.809, -31.975, 65.78, 38.02, -60.273]
  Call Extruder(262.38376)
  MoveL 9856 to (232.07, 163.02, 135.08) mm, rotated rx -180 ry 0 rz 180 deg; joints [-145.801, -75.775, -32.042, 65.76, 38.055, -60.239]
  MoveL 9857 to (232.07, 163.02, 135.08) mm, rotated rx -180 ry 0 rz 180 deg; joints [-145.801, -75.775, -32.042, 65.76, 38.055, -60.239]
  Call Extruder(262.56574)
  MoveL 9858 to (231.78, 163.15, 135.08) mm, rotated rx -180 ry 0 rz 180 deg; joints [-145.777, -75.742, -32.108, 65.741, 38.089, -60.205]
  MoveL 9859 to (231.78, 163.15, 135.08) mm, rotated rx -180 ry 0 rz 180 deg; joints [-145.777, -75.742, -32.108, 65.741, 38.089, -60.205]
  Call Extruder(262.71308)
  MoveL 9860 to (231.54, 163.24, 135.08) mm, rotated rx -180 ry 0 rz 180 deg; joints [-145.759, -75.714, -32.165, 65.723, 38.117, -60.175]
  MoveL 9861 to (231.54, 163.24, 135.08) mm, rotated rx -180 ry 0 rz 180 deg; joints [-145.759, -75.714, -32.165, 65.723, 38.117, -60.175]
  Call Extruder(262.82630)
  MoveL 9862 to (231.35, 163.3, 135.08) mm, rotated rx -180 ry 0 rz 180 deg; joints [-145.744, -75.69, -32.211, 65.708, 38.139, -60.15]
  MoveL 9863 to (231.35, 163.3, 135.08) mm, rotated rx -180 ry 0 rz 180 deg; joints [-145.744, -75.69, -32.211, 65.708, 38.139, -60.15]
  Call Extruder(262.93908)
  MoveL 9864 to (231.17, 163.36, 135.08) mm, rotated rx -180 ry 0 rz 180 deg; joints [-145.73, -75.667, -32.257, 65.693, 38.16, -60.125]
  MoveL 9865 to (231.17, 163.36, 135.08) mm, rotated rx -180 ry 0 rz 180 deg; joints [-145.73, -75.667, -32.257, 65.693, 38.16, -60.125]
  Call Extruder(263.05141)
  MoveL 9866 to (230.98, 163.42, 135.08) mm, rotated rx 180 ry 0 rz 180 deg; joints [-145.716, -75.644, -32.304, 65.677, 38.182, -60.1]
  MoveL 9867 to (230.98, 163.42, 135.08) mm, rotated rx 180 ry 0 rz 180 deg; joints [-145.716, -75.644, -32.304, 65.677, 38.182, -60.1]
  Call Extruder(263.16330)
  MoveL 9868 to (230.79, 163.48, 135.08) mm, rotated rx 180 ry 0 rz 180 deg; joints [-145.702, -75.62, -32.35, 65.662, 38.204, -60.075]
  MoveL 9869 to (230.79, 163.48, 135.08) mm, rotated rx 180 ry 0 rz 180 deg; joints [-145.702, -75.62, -32.35, 65.662, 38.204, -60.075]
  Call Extruder(263.28471)
  MoveL 9870 to (230.58, 163.55, 135.08) mm, rotated rx 180 ry 0 rz 180 deg; joints [-145.687, -75.595, -32.401, 65.645, 38.227, -60.048]
  MoveL 9871 to (230.58, 163.55, 135.08) mm, rotated rx 180 ry 0 rz 180 deg; joints [-145.687, -75.595, -32.401, 65.645, 38.227, -60.048]
  Call Extruder(263.41552)
  MoveL 9872 to (230.36, 163.61, 135.08) mm, rotated rx 180 ry 0 rz 180 deg; joints [-145.67, -75.567, -32.457, 65.626, 38.253, -60.017]
  MoveL 9873 to (230.36, 163.61, 135.08) mm, rotated rx 180 ry 0 rz 180 deg; joints [-145.67, -75.567, -32.457, 65.626, 38.253, -60.017]
  Call Extruder(263.54577)
  MoveL 9874 to (230.14, 163.68, 135.08) mm, rotated rx 180 ry 0 rz 180 deg; joints [-145.654, -75.539, -32.512, 65.607, 38.279, -59.987]
  MoveL 9875 to (230.14, 163.68, 135.08) mm, rotated rx 180 ry 0 rz 180 deg; joints [-145.654, -75.539, -32.512, 65.607, 38.279, -59.987]
  Call Extruder(263.67545)
  MoveL 9876 to (229.91, 163.75, 135.08) mm, rotated rx 180 ry 0 rz 180 deg; joints [-145.638, -75.511, -32.568, 65.589, 38.304, -59.957]
  MoveL 9877 to (229.91, 163.75, 135.08) mm, rotated rx 180 ry 0 rz 180 deg; joints [-145.638, -75.511, -32.568, 65.589, 38.304, -59.957]
  Call Extruder(263.80457)
  MoveL 9878 to (229.69, 163.82, 135.08) mm, rotated rx 180 ry 0 rz 180 deg; joints [-145.621, -75.483, -32.624, 65.57, 38.33, -59.926]
  MoveL 9879 to (229.69, 163.82, 135.08) mm, rotated rx 180 ry 0 rz 180 deg; joints [-145.621, -75.483, -32.624, 65.57, 38.33, -59.926]
  Call Extruder(263.91964)
  MoveL 9880 to (229.48, 163.86, 135.08) mm, rotated rx -180 ry 0 rz 180 deg; joints [-145.607, -75.456, -32.678, 65.55, 38.353, -59.895]
  MoveL 9881 to (229.48, 163.86, 135.08) mm, rotated rx -180 ry 0 rz 180 deg; joints [-145.607, -75.456, -32.678, 65.55, 38.353, -59.895]
  Call Extruder(264.03426)
  MoveL 9882 to (229.28, 163.91, 135.08) mm, rotated rx -180 ry 0 rz -180 deg; joints [-145.594, -75.428, -32.732, 65.53, 38.376, -59.865]
  MoveL 9883 to (229.28, 163.91, 135.08) mm, rotated rx -180 ry 0 rz -180 deg; joints [-145.594, -75.428, -32.732, 65.53, 38.376, -59.865]
  Call Extruder(264.14843)
  MoveL 9884 to (229.08, 163.95, 135.08) mm, rotated rx 180 ry 0 rz 180 deg; joints [-145.58, -75.401, -32.786, 65.51, 38.399, -59.834]
  MoveL 9885 to (229.08, 163.95, 135.08) mm, rotated rx 180 ry 0 rz 180 deg; joints [-145.58, -75.401, -32.786, 65.51, 38.399, -59.834]
  Call Extruder(264.26215)
  MoveL 9886 to (228.87, 164, 135.08) mm, rotated rx 180 ry 0 rz 180 deg; joints [-145.566, -75.374, -32.84, 65.491, 38.422, -59.803]
  MoveL 9887 to (228.87, 164, 135.08) mm, rotated rx 180 ry 0 rz 180 deg; joints [-145.566, -75.374, -32.84, 65.491, 38.422, -59.803]
  Call Extruder(264.38757)
  MoveL 9888 to (228.65, 164.04, 135.08) mm, rotated rx 180 ry 0 rz 180 deg; joints [-145.551, -75.344, -32.901, 65.468, 38.448, -59.769]
  MoveL 9889 to (228.65, 164.04, 135.08) mm, rotated rx 180 ry 0 rz 180 deg; joints [-145.551, -75.344, -32.901, 65.468, 38.448, -59.769]
  Call Extruder(264.52455)
  MoveL 9890 to (228.4, 164.09, 135.08) mm, rotated rx 180 ry 0 rz -180 deg; joints [-145.535, -75.31, -32.967, 65.444, 38.476, -59.731]
  MoveL 9891 to (228.4, 164.09, 135.08) mm, rotated rx 180 ry 0 rz -180 deg; joints [-145.535, -75.31, -32.967, 65.444, 38.476, -59.731]
  Call Extruder(264.66091)
  MoveL 9892 to (228.15, 164.14, 135.08) mm, rotated rx 180 ry 0 rz 180 deg; joints [-145.518, -75.277, -33.034, 65.419, 38.504, -59.692]
  MoveL 9893 to (228.15, 164.14, 135.08) mm, rotated rx 180 ry 0 rz 180 deg; joints [-145.518, -75.277, -33.034, 65.419, 38.504, -59.692]
  Call Extruder(264.79667)
  MoveL 9894 to (227.9, 164.19, 135.08) mm, rotated rx -180 ry 0 rz 180 deg; joints [-145.502, -75.243, -33.101, 65.394, 38.532, -59.654]
  MoveL 9895 to (227.9, 164.19, 135.08) mm, rotated rx -180 ry 0 rz 180 deg; joints [-145.502, -75.243, -33.101, 65.394, 38.532, -59.654]
  Call Extruder(264.93182)
  MoveL 9896 to (227.65, 164.24, 135.08) mm, rotated rx 180 ry 0 rz 180 deg; joints [-145.485, -75.21, -33.167, 65.37, 38.56, -59.616]
  MoveL 9897 to (227.65, 164.24, 135.08) mm, rotated rx 180 ry 0 rz 180 deg; joints [-145.485, -75.21, -33.167, 65.37, 38.56, -59.616]
  Call Extruder(265.06636)
  MoveL 9898 to (227.4, 164.29, 135.08) mm, rotated rx 180 ry 0 rz 180 deg; joints [-145.469, -75.176, -33.234, 65.346, 38.588, -59.579]
  MoveL 9899 to (227.4, 164.29, 135.08) mm, rotated rx 180 ry 0 rz 180 deg; joints [-145.469, -75.176, -33.234, 65.346, 38.588, -59.579]
  Call Extruder(265.20028)
  MoveL 9900 to (227.15, 164.34, 135.08) mm, rotated rx 180 ry 0 rz 180 deg; joints [-145.453, -75.143, -33.3, 65.321, 38.615, -59.541]
  MoveL 9901 to (227.15, 164.34, 135.08) mm, rotated rx 180 ry 0 rz 180 deg; joints [-145.453, -75.143, -33.3, 65.321, 38.615, -59.541]
  Call Extruder(265.34815)
  MoveL 9902 to (226.87, 164.39, 135.08) mm, rotated rx 180 ry 0 rz -180 deg; joints [-145.435, -75.106, -33.375, 65.294, 38.646, -59.498]
  MoveL 9903 to (226.87, 164.39, 135.08) mm, rotated rx 180 ry 0 rz -180 deg; joints [-145.435, -75.106, -33.375, 65.294, 38.646, -59.498]
  Call Extruder(265.50989)
  MoveL 9904 to (226.57, 164.44, 135.08) mm, rotated rx -180 ry 0 rz 180 deg; joints [-145.415, -75.064, -33.458, 65.262, 38.68, -59.45]
  MoveL 9905 to (226.57, 164.44, 135.08) mm, rotated rx -180 ry 0 rz 180 deg; joints [-145.415, -75.064, -33.458, 65.262, 38.68, -59.45]
  Call Extruder(265.67090)
  MoveL 9906 to (226.26, 164.49, 135.08) mm, rotated rx -180 ry 0 rz -180 deg; joints [-145.396, -75.022, -33.542, 65.231, 38.715, -59.402]
  MoveL 9907 to (226.26, 164.49, 135.08) mm, rotated rx -180 ry 0 rz -180 deg; joints [-145.396, -75.022, -33.542, 65.231, 38.715, -59.402]
  Call Extruder(265.83118)
  MoveL 9908 to (225.96, 164.54, 135.08) mm, rotated rx 180 ry 0 rz -180 deg; joints [-145.377, -74.98, -33.625, 65.199, 38.749, -59.354]
  MoveL 9909 to (225.96, 164.54, 135.08) mm, rotated rx 180 ry 0 rz -180 deg; joints [-145.377, -74.98, -33.625, 65.199, 38.749, -59.354]
  Call Extruder(265.99074)
  MoveL 9910 to (225.65, 164.58, 135.08) mm, rotated rx -180 ry 0 rz 180 deg; joints [-145.357, -74.938, -33.708, 65.168, 38.783, -59.306]
  MoveL 9911 to (225.65, 164.58, 135.08) mm, rotated rx -180 ry 0 rz 180 deg; joints [-145.357, -74.938, -33.708, 65.168, 38.783, -59.306]
  Call Extruder(266.14957)
  MoveL 9912 to (225.34, 164.63, 135.08) mm, rotated rx -180 ry 0 rz 180 deg; joints [-145.338, -74.897, -33.791, 65.138, 38.817, -59.259]
  MoveL 9913 to (225.34, 164.63, 135.08) mm, rotated rx -180 ry 0 rz 180 deg; joints [-145.338, -74.897, -33.791, 65.138, 38.817, -59.259]
  Call Extruder(266.32824)
  MoveL 9914 to (225, 164.68, 135.08) mm, rotated rx -180 ry 0 rz 180 deg; joints [-145.317, -74.849, -33.887, 65.101, 38.855, -59.203]
  MoveL 9915 to (225, 164.68, 135.08) mm, rotated rx -180 ry 0 rz 180 deg; joints [-145.317, -74.849, -33.887, 65.101, 38.855, -59.203]
  Call Extruder(266.52668)
  MoveL 9916 to (224.61, 164.72, 135.08) mm, rotated rx -180 ry 0 rz -180 deg; joints [-145.293, -74.795, -33.994, 65.06, 38.898, -59.141]
  MoveL 9917 to (224.61, 164.72, 135.08) mm, rotated rx -180 ry 0 rz -180 deg; joints [-145.293, -74.795, -33.994, 65.06, 38.898, -59.141]
  Call Extruder(266.72426)
  MoveL 9918 to (224.22, 164.77, 135.08) mm, rotated rx 180 ry 0 rz -180 deg; joints [-145.27, -74.741, -34.102, 65.019, 38.941, -59.078]
  MoveL 9919 to (224.22, 164.77, 135.08) mm, rotated rx 180 ry 0 rz -180 deg; joints [-145.27, -74.741, -34.102, 65.019, 38.941, -59.078]
  Call Extruder(266.92097)
  MoveL 9920 to (223.83, 164.82, 135.08) mm, rotated rx -180 ry 0 rz 180 deg; joints [-145.246, -74.687, -34.209, 64.978, 38.983, -59.016]
  MoveL 9921 to (223.83, 164.82, 135.08) mm, rotated rx -180 ry 0 rz 180 deg; joints [-145.246, -74.687, -34.209, 64.978, 38.983, -59.016]
  Call Extruder(267.11680)
  MoveL 9922 to (223.45, 164.86, 135.08) mm, rotated rx 180 ry 0 rz 180 deg; joints [-145.223, -74.633, -34.317, 64.938, 39.026, -58.954]
  MoveL 9923 to (223.45, 164.86, 135.08) mm, rotated rx 180 ry 0 rz 180 deg; joints [-145.223, -74.633, -34.317, 64.938, 39.026, -58.954]
  Call Extruder(267.41216)
  MoveL 9924 to (222.86, 164.91, 135.08) mm, rotated rx 180 ry 0 rz 180 deg; joints [-145.189, -74.549, -34.484, 64.873, 39.09, -58.856]
  MoveL 9925 to (222.86, 164.91, 135.08) mm, rotated rx 180 ry 0 rz 180 deg; joints [-145.189, -74.549, -34.484, 64.873, 39.09, -58.856]
  Call Extruder(267.70619)
  MoveL 9926 to (222.27, 164.96, 135.08) mm, rotated rx 180 ry 0 rz 180 deg; joints [-145.155, -74.466, -34.65, 64.808, 39.155, -58.758]
  MoveL 9927 to (222.27, 164.96, 135.08) mm, rotated rx 180 ry 0 rz 180 deg; joints [-145.155, -74.466, -34.65, 64.808, 39.155, -58.758]
  Call Extruder(267.99889)
  MoveL 9928 to (221.68, 165, 135.08) mm, rotated rx 180 ry 0 rz 180 deg; joints [-145.121, -74.383, -34.816, 64.744, 39.219, -58.662]
  MoveL 9929 to (221.68, 165, 135.08) mm, rotated rx 180 ry 0 rz 180 deg; joints [-145.121, -74.383, -34.816, 64.744, 39.219, -58.662]
  Call Extruder(268.57233)
  MoveL 9930 to (220.52, 165.05, 135.08) mm, rotated rx 180 ry 0 rz -180 deg; joints [-145.056, -74.215, -35.151, 64.612, 39.345, -58.464]
  MoveL 9931 to (220.52, 165.05, 135.08) mm, rotated rx 180 ry 0 rz -180 deg; joints [-145.056, -74.215, -35.151, 64.612, 39.345, -58.464]
  Call Extruder(269.28634)
  MoveL 9932 to (219.06, 165.09, 135.08) mm, rotated rx 180 ry 0 rz 180 deg; joints [-144.977, -74.005, -35.57, 64.448, 39.503, -58.217]
  Call Extruder(386.13307)
  MoveL 9933 to (-19.06, 165.09, 135.08) mm, rotated rx -180 ry 0 rz 180 deg; joints [-127.435, -52.868, -79.7, 62.623, 63.406, -40.843]
  Call Extruder(386.56168)
  MoveL 9934 to (-19.94, 165.07, 135.08) mm, rotated rx 180 ry 0 rz 180 deg; joints [-127.348, -52.819, -79.809, 62.67, 63.49, -40.816]
  MoveL 9935 to (-19.94, 165.07, 135.08) mm, rotated rx 180 ry 0 rz 180 deg; joints [-127.348, -52.819, -79.809, 62.67, 63.49, -40.816]
  Call Extruder(387.13513)
  MoveL 9936 to (-21.1, 165.03, 135.08) mm, rotated rx 180 ry 0 rz 180 deg; joints [-127.235, -52.753, -79.956, 62.73, 63.601, -40.778]
  MoveL 9937 to (-21.1, 165.03, 135.08) mm, rotated rx 180 ry 0 rz 180 deg; joints [-127.235, -52.753, -79.956, 62.73, 63.601, -40.778]
  Call Extruder(387.56943)
  MoveL 9938 to (-21.97, 164.98, 135.08) mm, rotated rx 180 ry 0 rz 180 deg; joints [-127.15, -52.702, -80.069, 62.774, 63.685, -40.748]
  MoveL 9939 to (-21.97, 164.98, 135.08) mm, rotated rx 180 ry 0 rz 180 deg; joints [-127.15, -52.702, -80.069, 62.774, 63.685, -40.748]
  Call Extruder(387.86345)
  MoveL 9940 to (-22.56, 164.93, 135.08) mm, rotated rx -180 ry 0 rz -180 deg; joints [-127.093, -52.667, -80.148, 62.802, 63.742, -40.727]
  MoveL 9941 to (-22.56, 164.93, 135.08) mm, rotated rx -180 ry 0 rz -180 deg; joints [-127.093, -52.667, -80.148, 62.802, 63.742, -40.727]
  Call Extruder(388.15881)
  MoveL 9942 to (-23.15, 164.89, 135.08) mm, rotated rx 180 ry 0 rz 180 deg; joints [-127.037, -52.632, -80.226, 62.831, 63.798, -40.705]
  MoveL 9943 to (-23.15, 164.89, 135.08) mm, rotated rx 180 ry 0 rz 180 deg; joints [-127.037, -52.632, -80.226, 62.831, 63.798, -40.705]
  Call Extruder(388.40503)
  MoveL 9944 to (-23.64, 164.84, 135.08) mm, rotated rx 180 ry 0 rz 180 deg; joints [-126.991, -52.602, -80.292, 62.854, 63.845, -40.686]
  MoveL 9945 to (-23.64, 164.84, 135.08) mm, rotated rx 180 ry 0 rz 180 deg; joints [-126.991, -52.602, -80.292, 62.854, 63.845, -40.686]
  Call Extruder(388.60173)
  MoveL 9946 to (-24.03, 164.79, 135.08) mm, rotated rx 180 ry 0 rz 180 deg; joints [-126.955, -52.578, -80.345, 62.871, 63.882, -40.67]
  MoveL 9947 to (-24.03, 164.79, 135.08) mm, rotated rx 180 ry 0 rz 180 deg; joints [-126.955, -52.578, -80.345, 62.871, 63.882, -40.67]
  Call Extruder(388.79931)
  MoveL 9948 to (-24.42, 164.75, 135.08) mm, rotated rx 180 ry 0 rz 180 deg; joints [-126.919, -52.554, -80.399, 62.889, 63.918, -40.654]
  MoveL 9949 to (-24.42, 164.75, 135.08) mm, rotated rx 180 ry 0 rz 180 deg; joints [-126.919, -52.554, -80.399, 62.889, 63.918, -40.654]
  Call Extruder(388.99775)
  MoveL 9950 to (-24.8, 164.7, 135.08) mm, rotated rx 180 ry 0 rz 180 deg; joints [-126.883, -52.53, -80.453, 62.906, 63.955, -40.638]
  MoveL 9951 to (-24.8, 164.7, 135.08) mm, rotated rx 180 ry 0 rz 180 deg; joints [-126.883, -52.53, -80.453, 62.906, 63.955, -40.638]
  Call Extruder(389.19706)
  MoveL 9952 to (-25.19, 164.66, 135.08) mm, rotated rx 180 ry 0 rz 180 deg; joints [-126.847, -52.506, -80.506, 62.924, 63.992, -40.622]
  MoveL 9953 to (-25.19, 164.66, 135.08) mm, rotated rx 180 ry 0 rz 180 deg; joints [-126.847, -52.506, -80.506, 62.924, 63.992, -40.622]
  Call Extruder(389.35589)
  MoveL 9954 to (-25.5, 164.61, 135.08) mm, rotated rx -180 ry 0 rz 180 deg; joints [-126.82, -52.487, -80.55, 62.937, 64.021, -40.608]
  MoveL 9955 to (-25.5, 164.61, 135.08) mm, rotated rx -180 ry 0 rz 180 deg; joints [-126.82, -52.487, -80.55, 62.937, 64.021, -40.608]
  Call Extruder(389.51545)
  MoveL 9956 to (-25.8, 164.56, 135.08) mm, rotated rx 180 ry 0 rz 180 deg; joints [-126.792, -52.467, -80.594, 62.949, 64.05, -40.594]
  MoveL 9957 to (-25.8, 164.56, 135.08) mm, rotated rx 180 ry 0 rz 180 deg; joints [-126.792, -52.467, -80.594, 62.949, 64.05, -40.594]
  Call Extruder(389.67574)
  MoveL 9958 to (-26.11, 164.51, 135.08) mm, rotated rx 180 ry 0 rz 180 deg; joints [-126.765, -52.447, -80.638, 62.962, 64.079, -40.58]
  MoveL 9959 to (-26.11, 164.51, 135.08) mm, rotated rx 180 ry 0 rz 180 deg; joints [-126.765, -52.447, -80.638, 62.962, 64.079, -40.58]
  Call Extruder(389.83676)
  MoveL 9960 to (-26.41, 164.46, 135.08) mm, rotated rx 180 ry 0 rz 180 deg; joints [-126.737, -52.428, -80.682, 62.975, 64.108, -40.566]
  MoveL 9961 to (-26.41, 164.46, 135.08) mm, rotated rx 180 ry 0 rz 180 deg; joints [-126.737, -52.428, -80.682, 62.975, 64.108, -40.566]
  Call Extruder(389.99850)
  MoveL 9962 to (-26.72, 164.41, 135.08) mm, rotated rx -180 ry 0 rz 180 deg; joints [-126.71, -52.408, -80.726, 62.988, 64.137, -40.553]
  MoveL 9963 to (-26.72, 164.41, 135.08) mm, rotated rx -180 ry 0 rz 180 deg; joints [-126.71, -52.408, -80.726, 62.988, 64.137, -40.553]
  Call Extruder(390.16097)
  MoveL 9964 to (-27.03, 164.36, 135.08) mm, rotated rx 180 ry 0 rz 180 deg; joints [-126.682, -52.388, -80.77, 63, 64.166, -40.539]
  MoveL 9965 to (-27.03, 164.36, 135.08) mm, rotated rx 180 ry 0 rz 180 deg; joints [-126.682, -52.388, -80.77, 63, 64.166, -40.539]
  Call Extruder(390.29490)
  MoveL 9966 to (-27.27, 164.32, 135.08) mm, rotated rx 180 ry 0 rz 180 deg; joints [-126.66, -52.372, -80.807, 63.01, 64.19, -40.526]
  MoveL 9967 to (-27.27, 164.32, 135.08) mm, rotated rx 180 ry 0 rz 180 deg; joints [-126.66, -52.372, -80.807, 63.01, 64.19, -40.526]
  Call Extruder(390.42943)
  MoveL 9968 to (-27.52, 164.27, 135.08) mm, rotated rx 180 ry 0 rz 180 deg; joints [-126.638, -52.355, -80.845, 63.019, 64.213, -40.514]
  MoveL 9969 to (-27.52, 164.27, 135.08) mm, rotated rx 180 ry 0 rz 180 deg; joints [-126.638, -52.355, -80.845, 63.019, 64.213, -40.514]
  Call Extruder(390.56458)
  MoveL 9970 to (-27.77, 164.22, 135.08) mm, rotated rx 180 ry 0 rz 180 deg; joints [-126.617, -52.338, -80.882, 63.029, 64.237, -40.501]
